(* CODESYS project OP60_PLC_program.project

Project tree, tasks and I/O mapping:
  Device : CODESYS Control Win V3 x64, 3S - Smart Software Solutions GmbH, version 3.5.16.40
    application Application
      libraries: VisuDialogs, * (System); MQTT Client SL, 1.0.2.0 (3S - Smart Software Solutions GmbH); SysTime, 3.5.9.0 (System); Util, * (System); StringUtils, 3.5.15.0 (System); Standard, * (System); SysFile, 3.5.15.0 (System)
      task MainTask (cyclic, interval t#20ms, priority 1) calls OP60_Main
      task AlarmManagerTask (cyclic, interval 50 ms, priority 1) calls AlarmManager.Alarm_Prg
      task VISU_TASK (cyclic, interval 100 ms, priority 1) calls VisuElems.Visu_Prg
      Symbols
      image pool ImagePool
      program SOP650 [LD]
      program OP60_Schedule [LD]
      FBs/
        function block FB_InputConveyor [LD]
        function block FB_SimpleConveyor [LD]
        function EraseSeconds [ST]
        program DateAndTime [ST]
        function TerminateString [ST]
        program CombineData [ST]
        function block FB_ModeControl [LD]
        function block FB_OutputConveyor [LD]
        function block FB_InspectionConveyor [LD]
        function Convert_RFID [ST]
      program SOP620 [LD]
      global variables GVL
      program OP60_Illumination [LD]
      program OP60_PublishMessages [LD]
      visualisation Production
      visualisation Overview
      program SOP690_GateEntry [LD]
      program OP60_Main [LD]
      program SOP600 [LD]
      program MQTTSub [ST]
      program SOP680 [LD]
      program SOP660 [LD]
      program Pruebas [LD]
      visualisation Manual_SOP640
      program SOP610 [LD]
      program SOP630 [LD]
      program OP60_Visu [LD]
      program MQTTPub [ST]
      visualisation Process
      visualisation Interfaces
      program SOP040_Safety [LD]
      global variables IOs
      Alarm Configuration
        alarm group SOP680_Alarms
            6814 [Fault]: Comparison Equal, ExpressionToCompare 14, Expression SOP680_FaultCode
            6805 [Fault]: Comparison Equal, ExpressionToCompare 5, Expression SOP680_FaultCode
            6811 [Fault]: Comparison Equal, ExpressionToCompare 11, Expression SOP680_FaultCode
            6802 [Fault]: Comparison Equal, ExpressionToCompare 2, Expression SOP680_FaultCode
            6812 [Fault]: Comparison Equal, ExpressionToCompare 12, Expression SOP680_FaultCode
            6810 [Fault]: Comparison Equal, ExpressionToCompare 10, Expression SOP680_FaultCode
            6801 [Fault]: Comparison Equal, ExpressionToCompare 1, Expression SOP680_FaultCode
            6813 [Fault]: Comparison Equal, ExpressionToCompare 13, Expression SOP680_FaultCode
        alarm class Fault (priority 10, acknowledge REP_ACK)
        alarm group SOP650_Alarms
            6512 [Fault]: Comparison Equal, ExpressionToCompare 12, Expression SOP650_FaultCode
            6514 [Fault]: Comparison Equal, ExpressionToCompare 14, Expression SOP650_FaultCode
            6501 [Fault]: Comparison Equal, ExpressionToCompare 1, Expression SOP650_FaultCode
            6511 [Fault]: Comparison Equal, ExpressionToCompare 11, Expression SOP650_FaultCode
            6510 [Fault]: Comparison Equal, ExpressionToCompare 10, Expression SOP650_FaultCode
            6505 [Fault]: Comparison Equal, ExpressionToCompare 5, Expression SOP650_FaultCode
            6513 [Fault]: Comparison Equal, ExpressionToCompare 13, Expression SOP650_FaultCode
            6502 [Fault]: Comparison Equal, ExpressionToCompare 2, Expression SOP650_FaultCode
        alarm group SOP660_Alarms
            6614 [Fault]: Comparison Equal, ExpressionToCompare 14, Expression SOP660_FaultCode
            6605 [Fault]: Comparison Equal, ExpressionToCompare 5, Expression SOP660_FaultCode
            6611 [Fault]: Comparison Equal, ExpressionToCompare 11, Expression SOP660_FaultCode
            6610 [Fault]: Comparison Equal, ExpressionToCompare 10, Expression SOP660_FaultCode
            6601 [Fault]: Comparison Equal, ExpressionToCompare 1, Expression SOP660_FaultCode
            6613 [Fault]: Comparison Equal, ExpressionToCompare 13, Expression SOP660_FaultCode
            6602 [Fault]: Comparison Equal, ExpressionToCompare 2, Expression SOP660_FaultCode
            6612 [Fault]: Comparison Equal, ExpressionToCompare 12, Expression SOP660_FaultCode
        alarm group SOP690_Alarms
            6901 [Fault]: Comparison Equal, ExpressionToCompare 0, Expression SOP690_NS1
            6902 [Fault]: Comparison Equal, ExpressionToCompare 0, Expression SOP690_B1
        alarm group SOP610_Alarms
            6110 [Fault]: Comparison Equal, ExpressionToCompare 10, Expression SOP610_FaultCode
            6101 [Fault]: Comparison Equal, ExpressionToCompare 1, Expression SOP610_FaultCode
            6111 [Fault]: Comparison Equal, ExpressionToCompare 11, Expression SOP610_FaultCode
            6114 [Fault]: Comparison Equal, ExpressionToCompare 14, Expression SOP610_FaultCode
            6105 [Fault]: Comparison Equal, ExpressionToCompare 5, Expression SOP610_FaultCode
            6113 [Fault]: Comparison Equal, ExpressionToCompare 13, Expression SOP610_FaultCode
            6102 [Fault]: Comparison Equal, ExpressionToCompare 2, Expression SOP610_FaultCode
            6112 [Fault]: Comparison Equal, ExpressionToCompare 12, Expression SOP610_FaultCode
        alarm group SOP670_Alarms
            6701 [Fault]: Comparison Equal, ExpressionToCompare 1, Expression SOP670_FaultCode
            6711 [Fault]: Comparison Equal, ExpressionToCompare 11, Expression SOP670_FaultCode
            6702 [Fault]: Comparison Equal, ExpressionToCompare 2, Expression SOP670_FaultCode
            6712 [Fault]: Comparison Equal, ExpressionToCompare 12, Expression SOP670_FaultCode
            6705 [Fault]: Comparison Equal, ExpressionToCompare 5, Expression SOP670_FaultCode
            6714 [Fault]: Comparison Equal, ExpressionToCompare 14, Expression SOP670_FaultCode
            6710 [Fault]: Comparison Equal, ExpressionToCompare 10, Expression SOP670_FaultCode
            6713 [Fault]: Comparison Equal, ExpressionToCompare 13, Expression SOP670_FaultCode
        alarm group SOP620_Alarms
            6205 [Fault]: Comparison Equal, ExpressionToCompare 5, Expression SOP620_FaultCode
            6202 [Fault]: Comparison Equal, ExpressionToCompare 2, Expression SOP620_FaultCode
            6212 [Fault]: Comparison Equal, ExpressionToCompare 12, Expression SOP620_FaultCode
            6201 [Fault]: Comparison Equal, ExpressionToCompare 1, Expression SOP620_FaultCode
            6211 [Fault]: Comparison Equal, ExpressionToCompare 11, Expression SOP620_FaultCode
            6213 [Fault]: Comparison Equal, ExpressionToCompare 13, Expression SOP620_FaultCode
            6210 [Fault]: Comparison Equal, ExpressionToCompare 10, Expression SOP620_FaultCode
            6214 [Fault]: Comparison Equal, ExpressionToCompare 14, Expression SOP620_FaultCode
        alarm group SOP600_Alarms
            6005 [Fault]: Comparison Equal, ExpressionToCompare 0, Expression SOP024_F12
            6003 [Fault]: Comparison Equal, ExpressionToCompare 0, Expression SOP024_F10
            6002 [Fault]: Comparison Equal, ExpressionToCompare 0, Expression SOP024_FQ1
            6008 [Fault]: Comparison Equal, ExpressionToCompare 0, Expression SOP040_B1
            6007 [Fault]: Comparison Equal, ExpressionToCompare 0, Expression SOP600_NS1
            6006 [Fault]: Comparison Equal, ExpressionToCompare 0, Expression SOP024_F13
            6004 [Fault]: Comparison Equal, ExpressionToCompare 0, Expression SOP024_F11
            6001 [Fault]: Comparison Equal, ExpressionToCompare 0, Expression SOP010_FQ1
        AlarmStorage
        alarm group SOP640_Alarms
            6402 [Fault]: Comparison Equal, ExpressionToCompare 2, Expression SOP640_FaultCode
            6412 [Fault]: Comparison Equal, ExpressionToCompare 12, Expression SOP640_FaultCode
            6422 [Fault]: Comparison Equal, ExpressionToCompare 22, Expression SOP640_FaultCode
            6410 [Fault]: Comparison Equal, ExpressionToCompare 10, Expression SOP640_FaultCode
            6414 [Fault]: Comparison Equal, ExpressionToCompare 14, Expression SOP640_FaultCode
            6413 [Fault]: Comparison Equal, ExpressionToCompare 13, Expression SOP640_FaultCode
            6420 [Fault]: Comparison Equal, ExpressionToCompare 20, Expression SOP640_FaultCode
            6430 [Fault]: Comparison Equal, ExpressionToCompare 0, Expression SOP640_LC1
            6405 [Fault]: Comparison Equal, ExpressionToCompare 5, Expression SOP640_FaultCode
            6401 [Fault]: Comparison Equal, ExpressionToCompare 1, Expression SOP640_FaultCode
            6411 [Fault]: Comparison Equal, ExpressionToCompare 11, Expression SOP640_FaultCode
            6421 [Fault]: Comparison Equal, ExpressionToCompare 21, Expression SOP640_FaultCode
            6423 [Fault]: Comparison Equal, ExpressionToCompare 23, Expression SOP640_FaultCode
        alarm class Warning (priority 30, acknowledge REP)
        text list TextList
        alarm group SOP630_Alarms
            6305 [Fault]: Comparison Equal, ExpressionToCompare 5, Expression SOP630_FaultCode
            6313 [Fault]: Comparison Equal, ExpressionToCompare 13, Expression SOP630_FaultCode
            6301 [Fault]: Comparison Equal, ExpressionToCompare 1, Expression SOP630_FaultCode
            6302 [Fault]: Comparison Equal, ExpressionToCompare 2, Expression SOP630_FaultCode
            6312 [Fault]: Comparison Equal, ExpressionToCompare 12, Expression SOP630_FaultCode
            6311 [Fault]: Comparison Equal, ExpressionToCompare 11, Expression SOP630_FaultCode
            6314 [Fault]: Comparison Equal, ExpressionToCompare 14, Expression SOP630_FaultCode
            6310 [Fault]: Comparison Equal, ExpressionToCompare 10, Expression SOP630_FaultCode
        alarm class Message (priority 100, acknowledge REP)
        alarm group OP60_Alarms
            0603 [Warning]: Comparison Equal, ExpressionToCompare 1, Expression OP60_ManDisInterlocks
            0601 [Message]: Comparison Equal, ExpressionToCompare 1, Expression OP60_WaitingToOP50
            0602 [Warning]: Comparison Equal, ExpressionToCompare 1, Expression OP60_EmptyMode
      program MQTT_Sensors_Actuators [LD]
      program SOP670 [LD]
      visualisation Diagnostics
      visualisation Manual_SOP610t630
      visualisation Manual_SOP650t680
      Cases/
        program Case1 [LD]
        program Case2 [LD]
        program Cases3_4_5 [LD]
      program SOP640 [LD]
  libraries: VisuSymbols, 3.5.10.0 (System)
  FuntionBlocks/
  5ce3da45-db07-42e7-a21c-a00fff4ed8f6|\\hsnas6\StaffHome\ayam\Documents\_MyStuff\13_Course AU334G\HMI\Motor Faulted.png
  visualisation Diagnostics
  5ce3da45-db07-42e7-a21c-a00fff4ed8f6|\\hsnas6\StaffHome\ayam\Documents\_MyStuff\13_Course AU334G\HMI\Door Open.png
  5ce3da45-db07-42e7-a21c-a00fff4ed8f6|\\hsnas6\StaffHome\ayam\Documents\_MyStuff\13_Course AU334G\HMI\Emergency Stop.png
  5ce3da45-db07-42e7-a21c-a00fff4ed8f6|\\hsnas6\StaffHome\ayam\Documents\_MyStuff\13_Course AU334G\HMI\Motor On.png
  5ce3da45-db07-42e7-a21c-a00fff4ed8f6|C:\Users\ayam\Dropbox\HiS\AUT02\Project\Layout.PNG
  5ce3da45-db07-42e7-a21c-a00fff4ed8f6|\\hsnas6\StaffHome\ayam\Documents\_MyStuff\13_Course AU334G\HMI\Motor Off.png
  text list GlobalTextList
  DataStructures/
    data type ProductionData
  text list System
  visualisation Production
  5ce3da45-db07-42e7-a21c-a00fff4ed8f6|\\hsnas6\StaffHome\ayam\Documents\_MyStuff\13_Course AU334G\HMI\Door Closed.png
*)

// DataStructures/ProductionData
TYPE ProductionData :
STRUCT
	ProductNr: UINT := 0; // Production Number
	IDNumber: UDINT := 0; // ID Number
	Status: WORD	:= 0; // Status Word
END_STRUCT
END_TYPE

// Device/Application/GVL
VAR_GLOBAL
	(* General *)
	Flash_1s: BOOL;		// Signal flashing (1Hz)
	Flash_2s: BOOL;		// Signal flashing (0.5Hz)
	Flash_2s_mem: BOOL;	// Flash_2s memory
	Client_Ready: BOOL;  // MQTT Ready
	ActualTime_hh_mm_ss: STRING; 		// Actual time HH:MM:SS format
	ActualTime_hh_mm: STRING;			// Actual time HH:MM:SS format
	Empty_PD : ProductionData;			// Empty Production Data
	
	Schedule_Start_msg: STRING(1024) := ''; 	// Received message from supervisor
	Schedule_End_msg: STRING(1024);		// Published message for supervisor
	Schedule_Start_msg_received: BOOL;		// Message is received again (this is made to avoid errors)
	Schedule_End_msg_received: BOOL; 			// Used to activate MQTT FB to publish message
	
	CycleData_Publish: BOOL; 				// Used to activate MQTT FB to publish message
	CycleData_pmsg: STRING(1024);			// Published message for further data analysis
	
	(* Light control should be in a sub-operation! *)
	Lights_msg: STRING(1024);			// Received message from supervisor/operator
	Lights_msg_received: BOOL;			// Message is received again (this is made to avoid errors)
	Switch_lights: BOOL;				// Used to activate turn on and off the lights
	Switch_msg: STRING(1024);			// Publish 'On' or 'Off' to turn on and off the lights
	Switch_publish: BOOL; 				// Order to publish
	Operator_pos_msg: STRING(1024);		// ????????????
	
	(* OP60 *)
	OP60_ModeControl: FB_ModeControl;
	OP60_Auto_On: BOOL; //OP60 in Auto-On
	OP60_Homing_On: BOOL; //OP60 in Homing-On
	OP60_Auto: BOOL; //OP60 in Auto Mode
	OP60_Manual: BOOL; // OP060 Manual Mode
	OP60_FaultAcc: BOOL; // OP60 Fault Accumulator
	OP60_WarningAcc: BOOL;	// OP60 Warning Accumulator
	OP60_SafetyCircuit_Ready: BOOL; // OP060 Safety Circuit Ready
	OP60_Stop_EOC_Req: BOOL; // OP060 Stop EOC Requested
	OP60_Stop_EOC_Ok: BOOL; // OP060 Stop EOC Ok
	OP60_HomePos_Ok: BOOL; // OP060 Home Position Ok
	OP60_ResetAlarms: BOOL; // OP60 Reset Alarms
	OP60_EOC AT %MW50: WORD; // OP060 EOC Word
	OP60_HomePos AT %MW51: WORD; // OP060 Home Pos Word
	OP60_ControlVoltage: BOOL; // Control Voltage Ready
	OP60_CtrlVoltageScheduleON: BOOL; // Control Voltage Schedule OFF
	OP60_CtrlVoltageScheduleOFF: BOOL; // Control Voltage Schedule ON
	OP60_WaitingToOP50: BOOL;	// OP60 Waiting to OP50
	OP60_WaitingToOP70: BOOL;	// OP60 Waiting to OP70
	OP60_ActualCycleTime: TIME; // Actual Cycle Time
	OP60_LastCycleTime: TIME; // Last Cycle Time
	OP60_TotalCycles: DWORD; // Total Cycles Counter
	OP60_EmptyMode: BOOL; // OP60 in Empty Mode
	OP60_ManDisInterlocks: BOOL; // OP060 Manual Mode
	OP60_ScheduleEnd: BOOL; // OP60 Schedule End
	OP60_ScheduleStart: BOOL; // OP60 Schedule Start
	HMI_DisableInterlocks: BOOL; // Disable Interlocks
	HMI_TotalCyclesReset: BOOL; //Total Cycles reset
	
	Operator_stop: BOOL;
	Operator_fault_msg: STRING(1024);
	Operator_fault_received: BOOL;
	
	SOP040_K1: BOOL;					// Safety Circuit OK
	SOP040_K1_msg: STRING(1024);		// OP60 Safety Circuit OK Message
	SOP040_K1_received: BOOL;			// Message is received again (this is made to avoid errors)
	SOP024_FQ1: BOOL;					// Power Suply Prim. Protection
	SOP024_FQ1_msg: STRING(1024);		// OP60 Power Suply Prim. Protection Message
	SOP024_FQ1_received: BOOL;			// Message is received again (this is made to avoid errors)
	SOP010_FQ1: BOOL;					// Supply Power Line Circuit Breaker
	SOP010_FQ1_msg: STRING(1024);		// OP60 Supply Power Line Circuit Breaker Message
	SOP010_FQ1_received: BOOL;			// Message is received again (this is made to avoid errors)
	SOP024_F10: BOOL;					// Power Suply Sec. Protection
	SOP024_F10_msg: STRING(1024);		// OP60 Power Suply Sec. Protection Message
	SOP024_F10_received: BOOL;			// Message is received again (this is made to avoid errors)
	SOP024_F11: BOOL;					// PLC Input Protection
	SOP024_F11_msg: STRING(1024);		// OP60 PLC Input Protection Message
	SOP024_F11_received: BOOL;			// Message is received again (this is made to avoid errors)
	SOP024_F12: BOOL;					// PLC Output Protection [HAY QUE QUITARLO]
	SOP024_F12_msg: STRING(1024);		// OP60 PLC Output Protection Message
	SOP024_F12_received: BOOL;			// Message is received again (this is made to avoid errors)
	SOP024_F13: BOOL;					// Safety Circuit Protection
	SOP024_F13_msg: STRING(1024);		// OP60 Safety Circuit Protection Message
	SOP024_F13_received: BOOL;			// Message is received again (this is made to avoid errors)
	SOP040_B1: BOOL;					// Pneumatic Pressure OK
	SOP040_B1_msg: STRING(1024);		// OP60 Pneumatic Pressure OK Message
	SOP040_B1_received: BOOL;			// Message is received again (this is made to avoid errors)
	
	(* OP50 Production Data *)
	OP50_PD : ProductionData;			// OP50 Last conveyor Production Data
	
	(* OP70 Production Data *)
	OP70_PD : ProductionData;			// OP70 First conveyor Production Data

	(* SOP600 *)
	SOP600_Faulted: BOOL;				// SOP600 Faulted
	
	SOP600_H1: BOOL;	// Control Voltage On Light
	SOP600_H2: BOOL; 	// Cycle Start Light
	SOP600_H3: BOOL;	// Cycle Stop Light
	SOP600_H4: BOOL; 	// Reset Alarm Light
	SOP600_H5: BOOL; 	// Reset Safety Light
	SOP600_H6: BOOL; 	// Blue Light
	SOP600_H7: BOOL; 	// Green Light
	SOP600_H8: BOOL; 	// Orange Light
	SOP600_H9: BOOL;	// Red Light
	SOP600_H10: BOOL;	// Home Position Light
	SOP600_H11: BOOL;	// Horn Sound
	
	SOP600_S1: BOOL;					// Control Voltage On
	SOP600_S1_msg: STRING(1024);		// SOP600_S1 Message
	SOP600_S1_received: BOOL;			// Message is received again (this is made to avoid errors)
	SOP600_S2: BOOL;					// Control Voltage Off
	SOP600_S2_msg: STRING(1024);		// SOP600_S2 Message
	SOP600_S2_received: BOOL;			// Message is received again (this is made to avoid errors)
	SOP600_S3: BOOL;					// Automatic Mode
	SOP600_S4: BOOL;					// Manual Mode
	SOP600_S3_4: BOOL;					// Automatic and Manual Mode
	SOP600_S3_4_msg: STRING(1024);		// SOP600_S4 Message
	SOP600_S3_4_received: BOOL;			// Message is received again (this is made to avoid errors)
	SOP600_S5: BOOL;					// Cycle Start
	SOP600_S5_msg: STRING(1024);		// SOP600_S5 Message
	SOP600_S5_received: BOOL;			// Message is received again (this is made to avoid errors)
	SOP600_S6: BOOL;					// Cycle Stop
	SOP600_S6_msg: STRING(1024);		// SOP600_S6 Message
	SOP600_S6_received: BOOL;			// Message is received again (this is made to avoid errors)
	SOP600_S7: BOOL;					// Halt
	SOP600_S7_msg: STRING(1024);		// SOP600_S7 Message
	SOP600_S7_received: BOOL;			// Message is received again (this is made to avoid errors)
	SOP600_S8: BOOL;					// Reset Alarm
	SOP600_S8_msg: STRING(1024);		// SOP600_S8 Message
	SOP600_S8_received: BOOL;			// Message is received again (this is made to avoid errors)
	SOP600_S9: BOOL;					// Reset Safety
	SOP600_S9_msg: STRING(1024);		// SOP600_S9 Message
	SOP600_S9_received: BOOL;			// Message is received again (this is made to avoid errors)
	SOP600_S10: BOOL;					// Home Position
	SOP600_S10_msg: STRING(1024);		// SOP600_S10 Message
	SOP600_S10_received: BOOL;			// Message is received again (this is made to avoid errors)
	SOP600_S11: BOOL;					// Emergency Stop
	SOP600_S11_msg: STRING(1024);		// SOP600_S11 Message
	SOP600_S11_received: BOOL;			// Message is received again (this is made to avoid errors)
	
	SOP040_K3: BOOL;					// Reset Safety circuit
	SOP040_K3_pmsg: STRING(1024);			// Published message for the logics
	SOP040_K3_publish: BOOL;				// Used to activate MQTT FB to publish message
	SOP600_H6_pmsg: STRING(1024);			// Published message for the logics
	SOP600_H6_publish: BOOL;				// Used to activate MQTT FB to publish message
	SOP600_H7_pmsg: STRING(1024);			// Published message for the logics
	SOP600_H7_publish: BOOL;				// Used to activate MQTT FB to publish message
	SOP600_H8_pmsg: STRING(1024);			// Published message for the logics
	SOP600_H8_publish: BOOL;				// Used to activate MQTT FB to publish message
	SOP600_H9_pmsg: STRING(1024);			// Published message for the logics
	SOP600_H9_publish: BOOL;				// Used to activate MQTT FB to publish message
	SOP600_S1_pmsg: STRING(1024);			// Published message for the logics
	SOP600_S1_publish: BOOL;				// Used to activate MQTT FB to publish message
	SOP600_S5_pmsg: STRING(1024);			// Published message for the logics
	SOP600_S5_publish: BOOL;				// Used to activate MQTT FB to publish message
	SOP600_S6_pmsg: STRING(1024);			// Published message for the logics
	SOP600_S6_publish: BOOL;				// Used to activate MQTT FB to publish message
	SOP600_S8_pmsg: STRING(1024);			// Published message for the logics
	SOP600_S8_publish: BOOL;				// Used to activate MQTT FB to publish message
	SOP600_S9_pmsg: STRING(1024);			// Published message for the logics
	SOP600_S9_publish: BOOL;				// Used to activate MQTT FB to publish message
	SOP600_S10_pmsg: STRING(1024);			// Published message for the logics
	SOP600_S10_publish: BOOL;				// Used to activate MQTT FB to publish message
	SOP600_S11_pmsg: STRING(1024);			// Published message for the logics
	SOP600_S11_publish: BOOL;				// Used to activate MQTT FB to publish message
	
	(* SOP610 *)
	SOP610_Conveyor: FB_InputConveyor; // SOP610_Conveyor
	SOP610_PD: ProductionData; 			// SOP610 Production Data
	SOP610_Faulted: BOOL;				// SOP610 Faulted
	SOP610_FaultCode: INT;				// SOP610 Fault Code
	SOP610_EOC AT %MX100.0: BOOL;		// SOP610 At EOC
	SOP610_HomePos AT %MX102.0: BOOL;	// SOP610 At Home Position
	
	SOP610_ReadyToTransfer: BOOL; 		// SOP610 Conveyor ready to transfer
	SOP610_Transfering: BOOL; 			// SOP610 Conveyor transfering
	SOP610_MovePD: BOOL;				// SOP610 Move Production Data
	
	HMI_SOP610_ManMoveFwd: BOOL; 		// SOP610 Manual Move Conveyor Fwd 
	HMI_SOP610_ManMoveRev: BOOL; 		// SOP610 Manual Move Conveyor Rev 
	HMI_SOP610_ManPDFwd: BOOL; 			// SOP610 Manual Move Production Data Fwd 
	HMI_SOP610_ManPDRev: BOOL; 			// SOP610 Manual Move Production Data Rev 
	
	SOP610_B1: BOOL;					// Conveyor Sensor
	SOP610_B1_msg: STRING(1024);		// SOP610 Photoelectric Sensor Message
	SOP610_B1_received: BOOL;			// Message is received again (this is made to avoid errors)
	SOP610_FQ1: BOOL;					// Motor Protection Tripped
	SOP610_FQ1_msg: STRING(1024);		// SOP610 Motor Protection Tripped Message
	SOP610_FQ1_received: BOOL;			// Message is received again (this is made to avoid errors)
	SOP610_RFID_Read: INT;							// RFID Read 
	SOP610_RFID_Read_msg: STRING(1024);				// SOP610 RFID Read Message
	SOP610_RFID_Read_received: BOOL;				// Message is received again (this is made to avoid errors)
	SOP610_RFID_Status: INT;						// RFID Status
	SOP610_RFID_Status_msg: STRING(1024);			// SOP610 RFID Status Message
	SOP610_RFID_Status_received: BOOL;				// Message is received again (this is made to avoid errors)
	
	// SOP610_RFID_Control: INT;				// RFID Contol
	SOP610_RFID_Control_pmsg: STRING(1024);	// Published message for the logics
	SOP610_RFID_Control_publish: BOOL;		// FB is publishing message
	// SOP610_RFID_Write: STRING;				// RFID Write
	SOP610_RFID_Write_pmsg: STRING(1024);	// Published message for the logics
	SOP610_RFID_Write_publish: BOOL;		// FB is publishing message
	SOP610_KM1: BOOL;						// Conveyor Forward
	SOP610_KM2: BOOL;						// Conveyor Reverse
	SOP610_KM1_2_pmsg: STRING(1024);		// Published message for the logics
	SOP610_KM1_2_pbusy: BOOL;				// FB is publishing message
	SOP610_KM1_2_publish: BOOL;				// Used to activate MQTT FB to publish message

	(* SOP620 *)
	SOP620_Conveyor: FB_SimpleConveyor; // SOP620_Conveyor
	SOP620_PD: ProductionData; 			// SOP620 Production Data
	SOP620_Faulted: BOOL;				// SOP620 Faulted
	SOP620_FaultCode: INT;				// SOP620 Fault Code
	SOP620_EOC AT %MX100.1: BOOL;		// SOP620 At EOC
	SOP620_HomePos AT %MX102.1: BOOL;	// SOP620 At Home Position
	
	SOP620_ReadyToTransfer: BOOL; 		// SOP620 Conveyor ready to transfer
	SOP620_Transfering: BOOL; 			// SOP620 Conveyor transfering
	SOP620_TransferOK: BOOL; 			// SOP620 Conveyor ready to load
	SOP620_TransferDone: BOOL; 			// SOP620 Conveyor load completed
	SOP620_MovePD: BOOL;				// SOP620 Move Production Data
	
	HMI_SOP620_ManMoveFwd: BOOL; 		// SOP620 Manual Move Conveyor Fwd 
	HMI_SOP620_ManMoveRev: BOOL; 		// SOP620 Manual Move Conveyor Rev 
	HMI_SOP620_ManPDFwd: BOOL; 			// SOP620 Manual Move Production Data Fwd 
	HMI_SOP620_ManPDRev: BOOL; 			// SOP620 Manual Move Production Data Rev 
	
	SOP620_B1: BOOL;					// Conveyor Sensor
	SOP620_B1_msg: STRING(1024);				// SOP620 Photoelectric Sensor Message
	SOP620_B1_received: BOOL;			// Message is received again (this is made to avoid errors)
	SOP620_FQ1: BOOL;					// Motor Protection Tripped
	SOP620_FQ1_msg: STRING(1024);		// SOP620 Motor Protection Tripped Message
	SOP620_FQ1_received: BOOL;			// Message is received again (this is made to avoid errors)
	
	SOP620_KM1: BOOL;						// Conveyor Forward
	SOP620_KM2: BOOL;						// Conveyor Reverse
	SOP620_KM1_2_pmsg: STRING(1024);		// Published message for the logics
	SOP620_KM1_2_pbusy: BOOL;				// FB is publishing message
	SOP620_KM1_2_publish: BOOL;				// Used to activate MQTT FB to publish message
	
	(* SOP630 *)
	SOP630_Conveyor: FB_SimpleConveyor; // SOP630_Conveyor
	SOP630_PD: ProductionData; 			// SOP630 Production Data
	SOP630_Faulted: BOOL;				// SOP630 Faulted
	SOP630_FaultCode: INT;				// SOP630 Fault Code
	SOP630_EOC AT %MX100.2: BOOL;		// SOP630 At EOC
	SOP630_HomePos AT %MX102.2: BOOL;	// SOP630 At Home Position
	
	SOP630_ReadyToTransfer: BOOL; 		// SOP630 Conveyor ready to transfer
	SOP630_Transfering: BOOL; 			// SOP630 Conveyor transfering
	SOP630_TransferOK: BOOL; 			// SOP630 Conveyor ready to load
	SOP630_TransferDone: BOOL; 			// SOP630 Conveyor load completed
	SOP630_MovePD: BOOL;				// SOP630 Move Production Data
	
	HMI_SOP630_ManMoveFwd: BOOL; 		// SOP630 Manual Move Conveyor Fwd 
	HMI_SOP630_ManMoveRev: BOOL; 		// SOP630 Manual Move Conveyor Rev 
	HMI_SOP630_ManPDFwd: BOOL; 			// SOP630 Manual Move Production Data Fwd 
	HMI_SOP630_ManPDRev: BOOL; 			// SOP630 Manual Move Production Data Rev 
	
	SOP630_B1: BOOL;					// Conveyor Sensor
	SOP630_B1_msg: STRING(1024);		// SOP630 Photoelectric Sensor Message
	SOP630_B1_received: BOOL;			// Message is received again (this is made to avoid errors)
	SOP630_FQ1: BOOL;					// Motor Protection Tripped
	SOP630_FQ1_msg: STRING(1024);		// SOP630 Motor Protection Tripped Message
	SOP630_FQ1_received: BOOL;			// Message is received again (this is made to avoid errors)
	
	SOP630_KM1: BOOL;						// Conveyor Forward
	SOP630_KM2: BOOL;						// Conveyor Reverse
	SOP630_KM1_2_pmsg: STRING(1024);		// Published message for the logics
	SOP630_KM1_2_pbusy: BOOL;				// FB is publishing message
	SOP630_KM1_2_publish: BOOL;				// Used to activate MQTT FB to publish message

	(* SOP640 *)
	SOP640_Conveyor: FB_InspectionConveyor; // SOP640_Conveyor
	SOP640_PD: ProductionData; 			// SOP640 Production Data
	SOP640_Faulted: BOOL;				// SOP640 Faulted
	SOP640_FaultCode: INT;				// SOP640 Fault Code
	SOP640_EOC AT %MX100.3: BOOL;		// SOP640 At EOC
	SOP640_HomePos AT %MX102.3: BOOL;	// SOP640 At Home Position
	
	SOP640_ReadyToTransfer: BOOL; 		// SOP640 Conveyor ready to transfer
	SOP640_Transfering: BOOL; 			// SOP640 Conveyor transfering
	SOP640_TransferOK: BOOL; 			// SOP640 Conveyor ready to load
	SOP640_TransferDone: BOOL; 			// SOP640 Conveyor load completed
	SOP640_MovePD: BOOL;				// SOP640 Move Production Data
	
	HMI_SOP640_ManMoveFwd: BOOL; 		// SOP640 Manual Move Conveyor Fwd 
	HMI_SOP640_ManMoveRev: BOOL; 		// SOP640 Manual Move Conveyor Rev 
	HMI_SOP640_ManFrontUp: BOOL;		// SOP640 Manual Move Front Clamp Up 
	HMI_SOP640_ManFrontDown: BOOL;		// SOP640 Manual Move Front Clamp Down
	HMI_SOP640_ManRearUp: BOOL;			// SOP640 Manual Move Rear Clamp Up
	HMI_SOP640_ManRearDown: BOOL;		// SOP640 Manual Move Rear Clamp Down
	HMI_SOP640_ManPDFwd: BOOL; 			// SOP640 Manual Move Production Data Fwd 
	HMI_SOP640_ManPDRev: BOOL; 			// SOP640 Manual Move Production Data Rev 
	HMI_SOP640_Accept: BOOL;			// SOP640 Accept Inspection
	HMI_SOP640_Discard: BOOL;			// SOP640 Discard Inspection
	HMI_SOP640_Inspecting: BOOL;		// SOP640 Discard Inspection
	
	SOP640_RS: BOOL;
	
	SOP640_Publish: BOOL; 				// Used to activate MQTT FB to publish message
	SOP640_pmsg: STRING(4096);			// Published message for operator
	SOP640_A1: BOOL;					// Conveyor Sensor
	SOP640_A1_msg: STRING(1024);		// SOP650 Photoelectric Sensor Message
	SOP640_A1_received: BOOL;			// Message is received again (this is made to avoid errors)
	SOP640_B1: BOOL;					// Conveyor Sensor
	SOP640_B1_msg: STRING(1024);				// SOP640 Photoelectric Sensor Message
	SOP640_B1_received: BOOL;			// Message is received again (this is made to avoid errors)
	SOP640_B2: BOOL(1024);					// Cylinder Sensor
	SOP640_B2_msg: STRING(1024);				// SOP640 Photoelectric Sensor Message
	SOP640_B2_received: BOOL;			// Message is received again (this is made to avoid errors)
	SOP640_B3: BOOL;					// Cylinder Sensor
	SOP640_B3_msg: STRING(1024);				// SOP640 Photoelectric Sensor Message
	SOP640_B3_received: BOOL;			// Message is received again (this is made to avoid errors)
	SOP640_B4: BOOL;					// Cylinder Sensor
	SOP640_B4_msg: STRING(1024);				// SOP640 Photoelectric Sensor Message
	SOP640_B4_received: BOOL;			// Message is received again (this is made to avoid errors)
	SOP640_B5: BOOL;					// Cylinder Sensor
	SOP640_B5_msg: STRING(1024);				// SOP640 Photoelectric Sensor Message
	SOP640_B5_received: BOOL;			// Message is received again (this is made to avoid errors)
	SOP640_B6: BOOL;					// Proximity Sensor
	SOP640_B6_msg: STRING(1024);				// SOP640 Photoelectric Sensor Message
	SOP640_B6_received: BOOL;			// Message is received again (this is made to avoid errors)
	SOP640_FQ1: BOOL;					// Motor Protection Tripped
	SOP640_FQ1_msg: STRING(1024);		// SOP640 Motor Protection Tripped Message
	SOP640_FQ1_received: BOOL;			// Message is received again (this is made to avoid errors)
	
	SOP640_KM1: BOOL;						// Conveyor Forward
	SOP640_KM2: BOOL;						// Conveyor Reverse
	SOP640_KM1_2_pmsg: STRING(1024);		// Published message for the logics
	SOP640_KM1_2_pbusy: BOOL;				// FB is publishing message
	SOP640_KM1_2_publish: BOOL;				// Used to activate MQTT FB to publish message
	SOP640_K2: BOOL;						// Stopper Up
	SOP640_K2_pmsg: STRING(1024);			// Published message for the logics
	SOP640_K2_publish: BOOL;				// Used to activate MQTT FB to publish message
	SOP640_Y1: BOOL;						// Stopper Up
	SOP640_Y1_pmsg: STRING(1024);			// Published message for the logics
	SOP640_Y1_publish: BOOL;				// Used to activate MQTT FB to publish message
	SOP640_Y2: BOOL;						// Stopper Down
	SOP640_Y2_pmsg: STRING(1024);			// Published message for the logics
	SOP640_Y2_publish: BOOL;				// Used to activate MQTT FB to publish message
	SOP640_Y3: BOOL;						// Stopper Up
	SOP640_Y3_pmsg: STRING(1024);			// Published message for the logics
	SOP640_Y3_publish: BOOL;				// Used to activate MQTT FB to publish message
	SOP640_Y4: BOOL;						// Stopper Down
	SOP640_Y4_pmsg: STRING(1024);			// Published message for the logics
	SOP640_Y4_publish: BOOL;				// Used to activate MQTT FB to publish message
	Products_publish: BOOL;					// Products data
	Products_pmsg: STRING(1024);			// Publish message for the logics
	
	// SOP640_RFID_Control: INT;				// RFID Contol
	SOP640_RFID_Control_pmsg: STRING(1024);	// Published message for the logics
	SOP640_RFID_Control_publish: BOOL;		// FB is publishing message
	// SOP640_RFID_Write: STRING;				// RFID Write
	SOP640_RFID_Write_pmsg: STRING(1024);	// Published message for the logics
	SOP640_RFID_Write_publish: BOOL;		// FB is publishing message
	
	Inspection_msg: STRING(1024) := ''; // Received message from SOP640 operator
	Inspection_msg_received: BOOL;		// Message is received again (this is made to avoid previous product status)

	(* SOP650 *)
	SOP650_Conveyor: FB_SimpleConveyor; // SOP650_Conveyor
	SOP650_PD: ProductionData; 			// SOP650 Production Data
	SOP650_Faulted: BOOL;				// SOP650 Faulted
	SOP650_FaultCode: INT;				// SOP650 Fault Code
	SOP650_EOC AT %MX100.4: BOOL;		// SOP650 At EOC
	SOP650_HomePos AT %MX102.4: BOOL;	// SOP650 At Home Position
	
	SOP650_ReadyToTransfer: BOOL; 		// SOP650 Conveyor ready to transfer
	SOP650_Transfering: BOOL; 			// SOP650 Conveyor transfering
	SOP650_TransferOK: BOOL; 			// SOP650 Conveyor ready to load
	SOP650_TransferDone: BOOL; 			// SOP650 Conveyor load completed
	SOP650_MovePD: BOOL;				// SOP650 Move Production Data
	
	HMI_SOP650_ManMoveFwd: BOOL; 		// SOP650 Manual Move Conveyor Fwd 
	HMI_SOP650_ManMoveRev: BOOL; 		// SOP650 Manual Move Conveyor Rev 
	HMI_SOP650_ManPDFwd: BOOL; 			// SOP650 Manual Move Production Data Fwd 
	HMI_SOP650_ManPDRev: BOOL; 			// SOP650 Manual Move Production Data Rev 
	
	
	SOP650_B1: BOOL;					// Conveyor Sensor
	SOP650_B1_msg: STRING(1024);		// SOP650 Photoelectric Sensor Message
	SOP650_B1_received: BOOL;			// Message is received again (this is made to avoid errors)
	SOP650_FQ1: BOOL;					// Motor Protection Tripped
	SOP650_FQ1_msg: STRING(1024);		// SOP610 Motor Protection Tripped Message
	SOP650_FQ1_received: BOOL;			// Message is received again (this is made to avoid errors)
	
	SOP650_KM1: BOOL;						// Conveyor Forward
	SOP650_KM2: BOOL;						// Conveyor Reverse
	SOP650_KM1_2_pbusy: BOOL;				// FB is publishing message
	SOP650_KM1_2_pmsg: STRING(1024);		// Published message for the logics
	SOP650_KM1_2_publish: BOOL;				// Used to activate MQTT FB to publish message

	(* SOP660 *)
	SOP660_Conveyor: FB_SimpleConveyor; // SOP660_Conveyor
	SOP660_PD: ProductionData; 			// SOP660 Production Data
	SOP660_Faulted: BOOL;				// SOP660 Faulted
	SOP660_FaultCode: INT;				// SOP660 Fault Code
	SOP660_EOC AT %MX100.5: BOOL;		// SOP660 At EOC
	SOP660_HomePos AT %MX102.5: BOOL;	// SOP660 At Home Position
	
	SOP660_ReadyToTransfer: BOOL; 		// SOP660 Conveyor ready to transfer
	SOP660_Transfering: BOOL; 			// SOP660 Conveyor transfering
	SOP660_TransferOK: BOOL; 			// SOP660 Conveyor ready to load
	SOP660_TransferDone: BOOL; 			// SOP660 Conveyor load completed
	SOP660_MovePD: BOOL;				// SOP660 Move Production Data
	
	HMI_SOP660_ManMoveFwd: BOOL; 		// SOP660 Manual Move Conveyor Fwd 
	HMI_SOP660_ManMoveRev: BOOL; 		// SOP660 Manual Move Conveyor Rev 
	HMI_SOP660_ManPDFwd: BOOL; 			// SOP660 Manual Move Production Data Fwd 
	HMI_SOP660_ManPDRev: BOOL; 			// SOP660 Manual Move Production Data Rev 
	
	SOP660_B1: BOOL;					// Conveyor Sensor
	SOP660_B1_msg: STRING(1024);		// SOP660 Photoelectric Sensor Message
	SOP660_B1_received: BOOL;			// Message is received again (this is made to avoid errors)
	SOP660_FQ1: BOOL;					// Motor Protection Tripped
	SOP660_FQ1_msg: STRING(1024);		// SOP660 Motor Protection Tripped Message
	SOP660_FQ1_received: BOOL;			// Message is received again (this is made to avoid errors)
	
	SOP660_KM1: BOOL;						// Conveyor Forward
	SOP660_KM2: BOOL;						// Conveyor Reverse
	SOP660_KM1_2_pbusy: BOOL;				// FB is publishing message
	SOP660_KM1_2_pmsg: STRING(1024);		// Published message for the logics
	SOP660_KM1_2_publish: BOOL;				// Used to activate MQTT FB to publish message

	(* SOP670 *)
	SOP670_Conveyor: FB_SimpleConveyor; // SOP670_Conveyor
	SOP670_PD: ProductionData; 			// SOP670 Production Data
	SOP670_Faulted: BOOL;				// SOP670 Faulted
	SOP670_FaultCode: INT;				// SOP670 Fault Code
	SOP670_EOC AT %MX100.6: BOOL;		// SOP670 At EOC
	SOP670_HomePos AT %MX102.6: BOOL;	// SOP670 At Home Position
	
	SOP670_ReadyToTransfer: BOOL; 		// SOP670 Conveyor ready to transfer
	SOP670_Transfering: BOOL; 			// SOP670 Conveyor transfering
	SOP670_TransferOK: BOOL; 			// SOP670 Conveyor ready to load
	SOP670_TransferDone: BOOL; 			// SOP670 Conveyor load completed
	SOP670_MovePD: BOOL;				// SOP670 Move Production Data
	
	HMI_SOP670_ManMoveFwd: BOOL; 		// SOP670 Manual Move Conveyor Fwd 
	HMI_SOP670_ManMoveRev: BOOL; 		// SOP670 Manual Move Conveyor Rev 
	HMI_SOP670_ManPDFwd: BOOL; 			// SOP670 Manual Move Production Data Fwd 
	HMI_SOP670_ManPDRev: BOOL; 			// SOP670 Manual Move Production Data Rev 
	
	SOP670_KM1: BOOL;						// Conveyor Forward
	SOP670_KM2: BOOL;						// Conveyor Reverse
	SOP670_KM1_2_pbusy: BOOL;				// FB is publishing message
	SOP670_B1: BOOL;					// Conveyor Sensor
	SOP670_B1_msg: STRING(1024);		// SOP670 Photoelectric Sensor Message
	SOP670_B1_received: BOOL;			// Message is received again (this is made to avoid errors)
	SOP670_FQ1: BOOL;					// Motor Protection Tripped
	SOP670_FQ1_msg: STRING(1024);		// SOP670 Motor Protection Tripped Message
	SOP670_FQ1_received: BOOL;			// Message is received again (this is made to avoid errors)
	
	SOP670_KM1_2_pmsg: STRING(1024);		// Published message for the logics
	SOP670_KM1_2_publish: BOOL;				// Used to activate MQTT FB to publish message

	(* SOP680 *)
	SOP680_Conveyor: FB_OutputConveyor; // SOP680_Conveyor
	SOP680_PD: ProductionData; 			// SOP680 Production Data
	SOP680_Faulted: BOOL;				// SOP680 Faulted
	SOP680_FaultCode: INT;				// SOP680 Fault Code
	SOP680_EOC AT %MX100.7: BOOL;		// SOP680 At EOC
	SOP680_HomePos AT %MX102.7: BOOL;	// SOP680 At Home Position
	
	SOP680_TransferOK: BOOL; 			// SOP680 Conveyor ready to load
	SOP680_TransferDone: BOOL; 			// SOP680 Conveyor load completed
	SOP680_MovePD: BOOL;				// SOP680 Move Production Data
	
	HMI_SOP680_ManMoveFwd: BOOL; 		// SOP680 Manual Move Conveyor Fwd 
	HMI_SOP680_ManMoveRev: BOOL; 		// SOP680 Manual Move Conveyor Rev 
	HMI_SOP680_ManPDFwd: BOOL; 			// SOP680 Manual Move Production Data Fwd 
	HMI_SOP680_ManPDRev: BOOL; 			// SOP680 Manual Move Production Data Rev 
	
	SOP680_B1: BOOL;					// Conveyor Sensor
	SOP680_B1_msg: STRING(1024);		// SOP680 Photoelectric Sensor Message
	SOP680_B1_received: BOOL;			// Message is received again (this is made to avoid errors)
	SOP680_FQ1: BOOL;					// Motor Protection Tripped
	SOP680_FQ1_msg: STRING(1024);		// SOP680 Motor Protection Tripped Message
	SOP680_FQ1_received: BOOL;			// Message is received again (this is made to avoid errors)
	
	SOP680_KM1: BOOL;						// Conveyor Forward
	SOP680_KM2: BOOL;						// Conveyor Reverse
	SOP680_KM1_2_pbusy: BOOL;				// FB is publishing message
	SOP680_KM1_2_pmsg: STRING(1024);		// Published message for the logics
	SOP680_KM1_2_publish: BOOL;				// Used to activate MQTT FB to publish message

	(* SOP690 *)
	SOP690_EntryRequest: BOOL;			// SOP690 Entry Request
	SOP690_Faulted: BOOL;				// SOP690 Faulted
	
	SOP690_K1: BOOL; 					// Gate Unlocked Confirmation
	SOP690_S1: BOOL;					// Cycle Start
	SOP690_S1_msg: STRING(1024);		// SOP690_S1 Message
	SOP690_S1_received: BOOL;			// Message is received again (this is made to avoid errors)
	SOP690_S2: BOOL;					// Entry Request
	SOP690_S2_msg: STRING(1024);		// SOP690_S2 Message
	SOP690_S2_received: BOOL;			// Message is received again (this is made to avoid errors)
	SOP690_S3: BOOL;					// Emergency Stop
	SOP690_S3_msg: STRING(1024);		// SOP690_S3 Message
	SOP690_S3_received: BOOL;			// Message is received again (this is made to avoid errors)
	SOP690_B1: BOOL;					// Gate Closed
	SOP690_S4: BOOL;					// Unlock Gate
	SOP690_S4_msg: STRING(1024);		// SOP690_S4 Message
	SOP690_S4_received: BOOL;			// Message is received again (this is made to avoid errors)

	SOP690_H1: BOOL;					// Cycle Start Light
	SOP690_H2: BOOL;					// Entry Request Light
	SOP690_H3: BOOL;					// Reset Safety Light
	
	SOP690_S1_pmsg: STRING(1024);			// Published message for the logics
	SOP690_S1_publish: BOOL;				// Used to activate MQTT FB to publish message
	SOP690_S2_pmsg: STRING(1024);			// Published message for the logics
	SOP690_S2_publish: BOOL;				// Used to activate MQTT FB to publish message
	SOP690_S3_pmsg: STRING(1024);			// Published message for the logics
	SOP690_S3_publish: BOOL;				// Used to activate MQTT FB to publish message
	SOP690_S4_pmsg: STRING(1024);			// Published message for the logics
	SOP690_S4_publish: BOOL;				// Used to activate MQTT FB to publish message
	
	SOP690_RFID_Read: INT;							// RFID Read 
	SOP690_RFID_Read_msg: STRING(1024);				// SOP690 RFID Read Message
	SOP690_RFID_Read_received: BOOL;				// Message is received again (this is made to avoid errors)
	SOP690_RFID_Status: INT;						// RFID Status
	SOP690_RFID_Status_msg: STRING(1024);			// SOP690 RFID Status Message
	SOP690_RFID_Status_received: BOOL;				// Message is received again (this is made to avoid errors)
	// SOP690_RFID_Control: INT;					// RFID Contol
	SOP690_RFID_Control_pmsg: STRING(1024);			// Published message for the logics
	SOP690_RFID_Control_publish: BOOL;				// FB is publishing message
END_VAR

// Device/Application/IOs
VAR_GLOBAL
	(* INPUTS*) 
	//Name	Address	Type	Comment
	SOP004_A1_4	AT %MW0	: WORD;	// 16 DI Card, Input 0-7 
	//1 SOP010_FQ1	AT %MX0.0	: BOOL;	// Supply Power Line Circuit Breaker
	//2 SOP040_K1	AT %MX0.1	: BOOL;	// Safety Circuit OK
	//3 SOP024_FQ1	AT %MX0.2	: BOOL;	// Power Suply Prim. Protection
	//4 SOP024_F10	AT %MX0.3	: BOOL;	// Power Suply Sec. Protection
	//5 SOP024_F11	AT %MX0.4	: BOOL;	// PLC Input Protection
	//6 SOP024_F12	AT %MX0.5	: BOOL;	// PLC Output Protection
	//7 SOP024_F13	AT %MX0.6	: BOOL;	// Safety Circuit Protection
	//8 SOP040_B1	AT %MX0.7	: BOOL;	// Pneumatic Pressure OK
	//SOP004_A1_4_2	AT %MB1	: BYTE;	// 16 DI Card, Input 8-15 
	M16_Entry	AT %MX1.0	: BOOL;	// 
	M16T_Entry	AT %MX1.1	: BOOL;	// 
	M20_Entry	AT %MX1.2	: BOOL;	// 
	M24_Entry	AT %MX1.3	: BOOL;	// 
	//Reserved	AT %MX1.4	: BOOL;	// 
	//Reserved	AT %MX1.5	: BOOL;	// 
	//Reserved	AT %MX1.6	: BOOL;	// 
	//Reserved	AT %MX1.7	: BOOL;	// 
	SOP004_A1_5	AT %MW1	: WORD;	// 16 DI Card, Input 0-7 
	//9 SOP600_S1	AT %MX2.0	: BOOL;	// Control Voltage On
	//10 SOP600_S2	AT %MX2.1	: BOOL;	// Control Voltage Off
	//11 SOP600_S3	AT %MX2.2	: BOOL;	// Manual Mode
	//12 SOP600_S4	AT %MX2.3	: BOOL;	// Automatic Mode
	//13 SOP600_S5	AT %MX2.4	: BOOL;	// Cycle Start
	//14 SOP600_S6	AT %MX2.5	: BOOL;	// Cycle Stop
	//15 SOP600_S7	AT %MX2.6	: BOOL;	// Halt
	//16 SOP600_S8	AT %MX2.7	: BOOL;	// Reset Alarm
	//SOP004_A1_5_2	AT %MB3	: BYTE;	// 16 DI Card, Input 8-15 
	//17 SOP600_S9	AT %MX3.0	: BOOL;	// Reset Safety
	//18 SOP600_S10	AT %MX3.1	: BOOL;	// Home Position     (* SOP600_S11 NOT DEFINED? *)
	SOP600_NS1	AT %MX3.2	: BOOL;	// Emergency Stop
	//Reserved	AT %MX3.3	: ;	// 
	//Reserved	AT %MX3.4	: ;	// 
	//Reserved	AT %MX3.5	: ;	// 
	//Reserved	AT %MX3.6	: ;	// 
	//Reserved	AT %MX3.7	: ;	// 
	SOP004_A1_6	AT %MW2	: WORD;	// 16 DI Card, Input 0-7 
	//19 SOP610_FQ1	AT %MX4.0	: BOOL;	// Motor Protection Tripped
	//20 SOP610_B1	AT %MX4.1	: BOOL;	// Conveyor Sensor
	//21 SOP620_FQ1	AT %MX4.2	: BOOL;	// Motor Protection Tripped
	//22 SOP620_B1	AT %MX4.3	: BOOL;	// Conveyor Sensor
	//23 SOP630_FQ1	AT %MX4.4	: BOOL;	// Motor Protection Tripped
	//24 SOP630_B1	AT %MX4.5	: BOOL;	// Conveyor Sensor
	//Reserved	AT %MX4.6	: ;	// 
	//Reserved	AT %MX4.7	: ;	// 
	//SOP004_A1_6_2	AT %MB5	: BYTE;	// 16 DI Card, Input 8-15 
	//25 SOP640_FQ1	AT %MX5.0	: BOOL;	// Motor Protection Tripped
	//26 SOP640_B1	AT %MX5.1	: BOOL;	// Conveyor Sensor
	//27 SOP640_B2	AT %MX5.2	: BOOL;	// Front Clamp Down
	//28 SOP640_B3	AT %MX5.3	: BOOL;	// Front Clamp Up
	//29 SOP640_B4	AT %MX5.4	: BOOL;	// Rear Clamp Down
	//30 SOP640_B5	AT %MX5.5	: BOOL;	// Rear Clamp Up
	//31 SOP640_B6	AT %MX5.6	: BOOL;	// Operator Proximity Sensor 
	SOP640_LC1	AT %MX5.7	: BOOL;	// Light Curtain OK
	SOP004_A1_7	AT %MW3	: WORD;	// 16 DI Card, Input 0-7 
	//33 SOP650_FQ1	AT %MX6.0	: BOOL;	// Motor Protection Tripped
	//34 SOP650_B1	AT %MX6.1	: BOOL;	// Conveyor Sensor
	//35 SOP660_FQ1	AT %MX6.2	: BOOL;	// Motor Protection Tripped
	//36 SOP660_B1	AT %MX6.3	: BOOL;	// Conveyor Sensor
	//37 SOP670_FQ1	AT %MX6.4	: BOOL;	// Motor Protection Tripped
	//38 SOP670_B1	AT %MX6.5	: BOOL;	// Conveyor Sensor
	//39 SOP680_FQ1	AT %MX6.6	: BOOL;	// Motor Protection Tripped
	//40 SOP680_B1	AT %MX6.7	: BOOL;	// Conveyor Sensor
	//SOP004_A1_7_2	AT %MB7	: BYTE;	// 16 DI Card, Input 8-15 
	//Reserved	AT %MX7.0	: BOOL;	// 
	//Reserved	AT %MX7.1	: BOOL;	// 
	//Reserved	AT %MX7.2	: BOOL;	// 
	//Reserved	AT %MX7.3	: BOOL;	// 
	//Reserved	AT %MX7.4	: BOOL;	// 
	//Reserved	AT %MX7.5	: BOOL;	// 
	//Reserved	AT %MX7.6	: BOOL;	// 
	//Reserved	AT %MX7.7	: BOOL;	// 
	SOP004_A3_2	AT %MW4	: WORD;	// 16 DI Card, Input 0-7 
	//41 SOP690_S1	AT %MX8.0	: BOOL;	// Cycle Start
	//42 SOP690_S2	AT %MX8.1	: BOOL;	// Entry Request
	//43 SOP690_S3	AT %MX8.2	: BOOL;	// Reset Safety
	SOP690_NS1	AT %MX8.3	: BOOL;	// Emergency Stop
	//Reserved	AT %MX8.4	: BOOL;	// 
	//Reserved	AT %MX8.5	: BOOL;	// 
	//Reserved	AT %MX8.6	: BOOL;	// 
	//Reserved	AT %MX8.7	: BOOL;	// 
	//SOP004_A3_2_2	AT %MB9	: BYTE;	// 16 DI Card, Input 8-15 
	//44 SOP690_K1	AT %MX9.0	: BOOL;	// Gate Unlocked Confirmation
    //45 SOP690_B1	AT %MX9.1	: BOOL;	// Gate Closed
	//Reserved	AT %MX9.2	: BOOL;	// 
	//Reserved	AT %MX9.3	: BOOL;	// 
	//Reserved	AT %MX9.4	: BOOL;	// 
	//Reserved	AT %MX9.5	: BOOL;	// 
	//Reserved	AT %MX9.6	: BOOL;	// 
	//Reserved	AT %MX9.7	: BOOL;	// 

	(* OUTPUTS *)
	SOP004_A1_8	AT %QW0	: WORD;	// 16 DO Card, Output 0-7 
    //46 SOP040_K3	AT %QX0.0	: BOOL;	// Reset Safety circuit // Por declarar
	SOP040_K4	AT %QX0.1	: BOOL;	// Safety Power Line
	SOP040_K5	AT %QX0.2	: BOOL;	// Safety Pneumatics
	//Reserved	AT %QX0.3	: BOOL;	// 
	//Reserved	AT %QX0.4	: BOOL;	// 
	//47 SOP600_H1	AT %QX0.5	: BOOL;	// Control Voltage On Light
	//48 SOP600_H2	AT %QX0.6	: BOOL;	// Cycle Start Light
	//49 SOP600_H3	AT %QX0.7	: BOOL;	// Cycle Stop Light
	//SOP004_A1_8_2	AT %QB1	: BYTE;	// 16 DO Card, Output 8-15 
	//50 SOP600_H4	AT %QX1.0	: BOOL;	// Reset Alarm Light
	//51 SOP600_H5	AT %QX1.1	: BOOL;	// Reset Safety Light
	//52 SOP600_H6	AT %QX1.2	: BOOL;	// Blue Light
	//53 SOP600_H7	AT %QX1.3	: BOOL;	// Green Light
	//54 SOP600_H8	AT %QX1.4	: BOOL;	// Orange Light
	//55 SOP600_H9	AT %QX1.5	: BOOL;	// Red Light
	//56 SOP600_H10	AT %QX1.6	: BOOL;	// Home Position Light
	//57 SOP600_H11	AT %QX1.7	: BOOL;	// Horn sound
	SOP004_A1_9	AT %QW1	: WORD;	// 16 DO Card, Output 0-7 
	//58 SOP610_KM1	AT %QX2.0	: BOOL;	// Conveyor Forward
	//59 SOP610_KM2	AT %QX2.1	: BOOL;	// Conveyor Reverse
	//60 SOP620_KM1	AT %QX2.2	: BOOL;	// Conveyor Forward
	//61 SOP620_KM2	AT %QX2.3	: BOOL;	// Conveyor Reverse
	//62 SOP630_KM1	AT %QX2.4	: BOOL;	// Conveyor Forward
	//63 SOP630_KM2	AT %QX2.5	: BOOL;	// Conveyor Reverse
	//Reserved	AT %QX2.6	: BOOL;	// 
	//Reserved	AT %QX2.7	: BOOL;	// 
	//SOP004_A1_9_2	AT %QB3	: BYTE;	// 16 DO Card, Output 8-15 
	//64 SOP640_KM1	AT %QX3.0	: BOOL;	// Conveyor Forward
	//65 SOP640_KM2	AT %QX3.1	: BOOL;	// Conveyor Reverse
	//66 SOP640_Y1	AT %QX3.2	: BOOL;	// Front Clamp Up
	//67 SOP640_Y2	AT %QX3.3	: BOOL;	// Front Clamp Down
	//68 SOP640_Y3	AT %QX3.4	: BOOL;	// Rear Clamp Up
	//69 SOP640_Y4	AT %QX3.5	: BOOL;	// Rear Clamp Down
	//Reserved	AT %QX3.6	: BOOL;	// 
	//70 SOP640_K2	AT %QX3.7	: BOOL;	// Light Curtain Muting 
	SOP004_A1_10	AT %QW2	: WORD;	// 16 DO Card, Output 0-7 
	//71 SOP650_KM1	AT %QX4.0	: BOOL;	// Conveyor Forward
	//72 SOP650_KM2	AT %QX4.1	: BOOL;	// Conveyor Reverse
	//73 SOP660_KM1	AT %QX4.2	: BOOL;	// Conveyor Forward
	//74 SOP660_KM2	AT %QX4.3	: BOOL;	// Conveyor Reverse
	//75 SOP670_KM1	AT %QX4.4	: BOOL;	// Conveyor Forward
	//76 SOP670_KM2	AT %QX4.5	: BOOL;	// Conveyor Reverse
	//77 SOP680_KM1	AT %QX4.6	: BOOL;	// Conveyor Forward
	//78 SOP680_KM2	AT %QX4.7	: BOOL;	// Conveyor Reverse
	//SOP004_A1_10_2	AT %QB5	: BYTE;	// 16 DO Card, Output 8-15 
	//Reserved	AT %QX5.0	: BOOL;	// 
	//Reserved	AT %QX5.1	: BOOL;	// 
	//Reserved	AT %QX5.2	: BOOL;	// 
	//Reserved	AT %QX5.3	: BOOL;	// 
	//Reserved	AT %QX5.4	: BOOL;	// 
	//Reserved	AT %QX5.5	: BOOL;	// 
	//Reserved	AT %QX5.6	: BOOL;	// 
	//Reserved	AT %QX5.7	: BOOL;	// 
	SOP004_A3_3	AT %QW3	: WORD;	// 16 DO Card, Output 0-7 
	//79 SOP690_H1	AT %QX6.0	: BOOL;	// Cycle Start Light
	//80 SOP690_H2	AT %QX6.1	: BOOL;	// Entry Request Light
	//81 SOP690_H3	AT %QX6.2	: BOOL;	// Reset Safety Light
	//Reserved	AT %QX6.3	: BOOL;	// 
	//Reserved	AT %QX6.4	: BOOL;	// 
	//Reserved	AT %QX6.5	: BOOL;	// 
	//Reserved	AT %QX6.6	: BOOL;	// 
	//Reserved	AT %QX6.7	: BOOL;	// 
	//SOP004_A3_3_2	AT %QB7	: BYTE;	// 16 DO Card, Output 8-15 
	//82 SOP690_S4	AT %QX7.0	: BOOL;	// Unlock Gate
	//Reserved	AT %QX7.1	: BOOL;	// 
	//Reserved	AT %QX7.2	: BOOL;	// 
	//Reserved	AT %QX7.3	: BOOL;	// 
	//Reserved	AT %QX7.4	: BOOL;	// 
	//Reserved	AT %QX7.5	: BOOL;	// 
	//Reserved	AT %QX7.6	: BOOL;	// 
	//Reserved	AT %QX7.7	: BOOL;	// 	
END_VAR

// Device/Application/OP60_Main
PROGRAM OP60_Main
VAR
	
	RS_0: RS;
	Operator_Faulted: BOOL;
	RS_1: RS;
	Stop: BOOL;
END_VAR
VAR // added by the converter: edge detectors and wires of the graphical bodies
    _rt1, _rt2, _rt3 : R_TRIG;
    _w1, _w2, _w3, _w4 : BOOL;
    _ft1, _ft2 : F_TRIG;
END_VAR

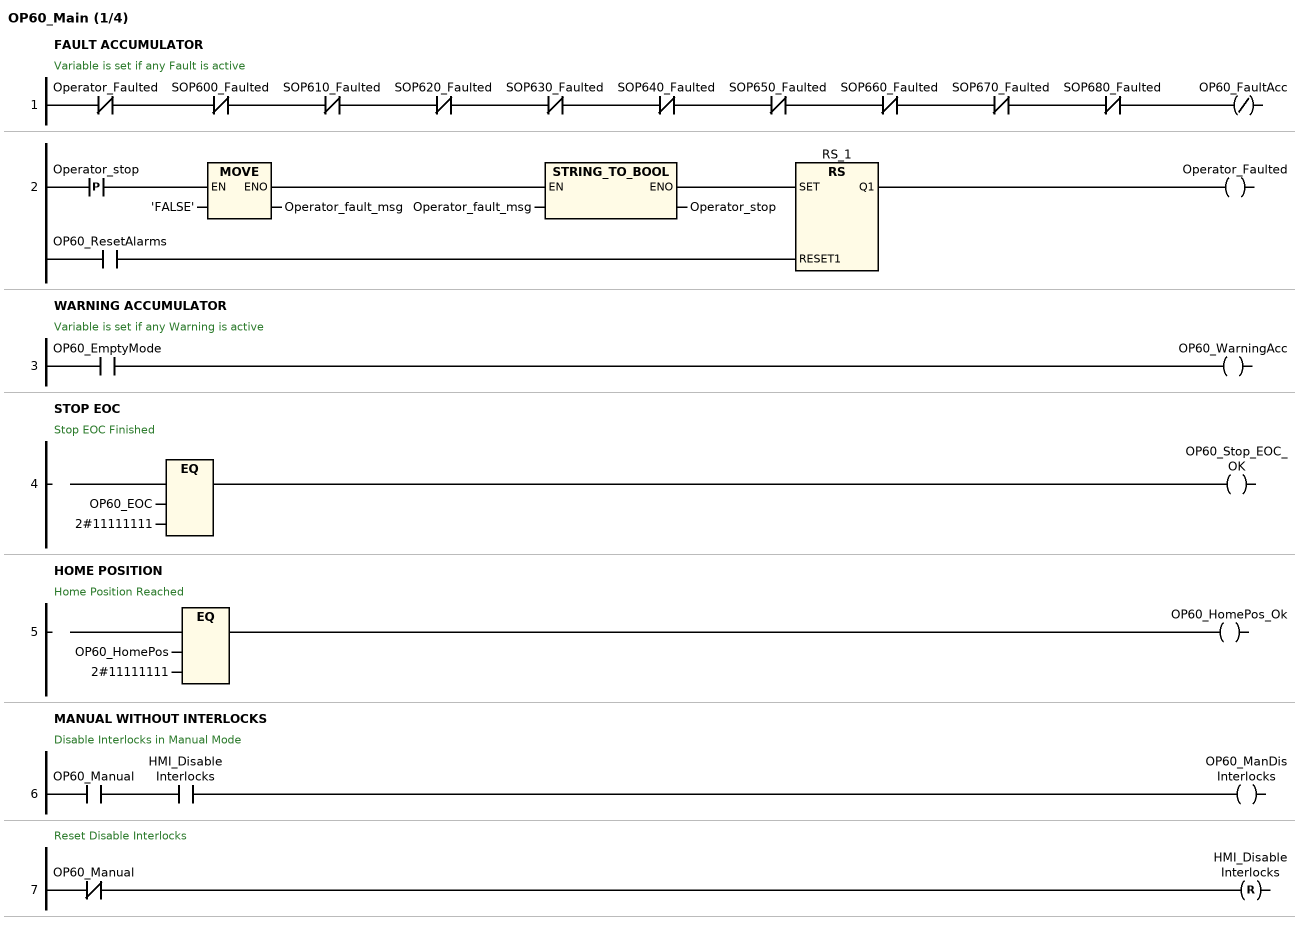
// NETWORK 1: FAULT ACCUMULATOR
// Variable is set if any Fault is active
OP60_FaultAcc := NOT (NOT Operator_Faulted AND NOT SOP600_Faulted AND NOT SOP610_Faulted AND NOT SOP620_Faulted AND NOT SOP630_Faulted AND NOT SOP640_Faulted AND NOT SOP650_Faulted AND NOT SOP660_Faulted AND NOT SOP670_Faulted AND NOT SOP680_Faulted);

// NETWORK 2
_rt1(CLK := Operator_stop);
_w1 := _rt1.Q;
IF _w1 THEN Operator_fault_msg := 'FALSE'; END_IF
IF _w1 THEN Operator_stop := STRING_TO_BOOL(Operator_fault_msg); END_IF
RS_1(SET := _w1, RESET1 := OP60_ResetAlarms); // RS
Operator_Faulted := RS_1.Q1;

// NETWORK 3: WARNING ACCUMULATOR
// Variable is set if any Warning is active
OP60_WarningAcc := OP60_EmptyMode;

// NETWORK 4: STOP EOC
// Stop EOC Finished
OP60_Stop_EOC_OK := OP60_EOC = 2#11111111;

// NETWORK 5: HOME POSITION
// Home Position Reached
OP60_HomePos_Ok := OP60_HomePos = 2#11111111;

// NETWORK 6: MANUAL WITHOUT INTERLOCKS
// Disable Interlocks in Manual Mode
OP60_ManDisInterlocks := OP60_Manual AND HMI_DisableInterlocks;

// NETWORK 7
// Reset Disable Interlocks
HMI_DisableInterlocks R= NOT OP60_Manual;

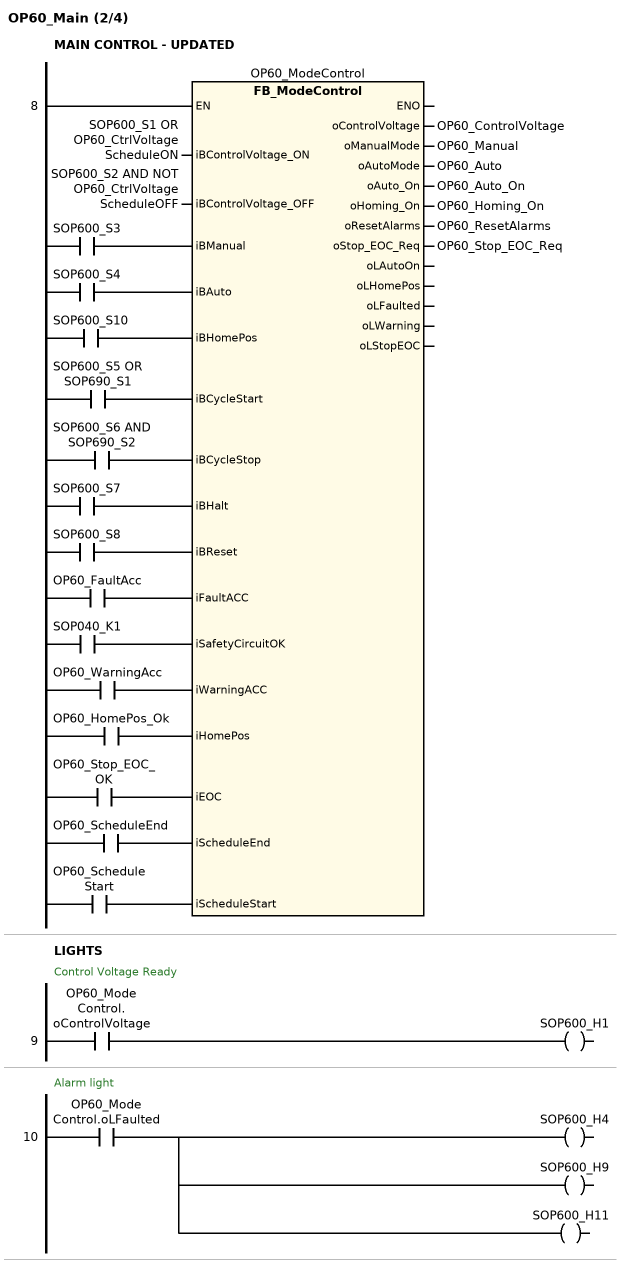
// NETWORK 8: MAIN CONTROL - UPDATED
OP60_ModeControl(
    iBControlVoltage_ON := SOP600_S1 OR OP60_CtrlVoltageScheduleON,
    iBControlVoltage_OFF := SOP600_S2 AND NOT OP60_CtrlVoltageScheduleOFF,
    iBManual := SOP600_S3,
    iBAuto := SOP600_S4,
    iBHomePos := SOP600_S10,
    iBCycleStart := SOP600_S5 OR SOP690_S1,
    iBCycleStop := SOP600_S6 AND SOP690_S2,
    iBHalt := SOP600_S7,
    iBReset := SOP600_S8,
    iFaultACC := OP60_FaultAcc,
    iSafetyCircuitOK := SOP040_K1,
    iWarningACC := OP60_WarningAcc,
    iHomePos := OP60_HomePos_Ok,
    iEOC := OP60_Stop_EOC_OK,
    iScheduleEnd := OP60_ScheduleEnd,
    iScheduleStart := OP60_ScheduleStart,
    oControlVoltage => OP60_ControlVoltage,
    oManualMode => OP60_Manual,
    oAutoMode => OP60_Auto,
    oAuto_On => OP60_Auto_On,
    oHoming_On => OP60_Homing_On,
    oResetAlarms => OP60_ResetAlarms,
    oStop_EOC_Req => OP60_Stop_EOC_Req); // FB_ModeControl

// NETWORK 9: LIGHTS
// Control Voltage Ready
SOP600_H1 := OP60_ModeControl.oControlVoltage;

// NETWORK 10
// Alarm light
SOP600_H4 := OP60_ModeControl.oLFaulted;
SOP600_H9 := OP60_ModeControl.oLFaulted;
SOP600_H11 := OP60_ModeControl.oLFaulted;

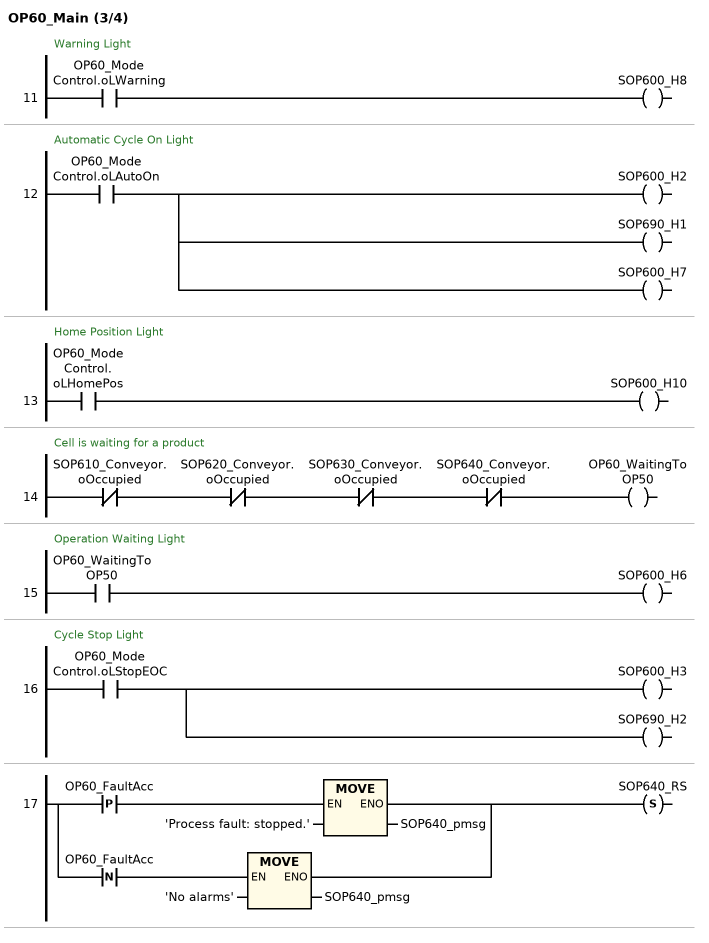
// NETWORK 11
// Warning Light
SOP600_H8 := OP60_ModeControl.oLWarning;

// NETWORK 12
// Automatic Cycle On Light
SOP600_H2 := OP60_ModeControl.oLAutoOn;
SOP690_H1 := OP60_ModeControl.oLAutoOn;
SOP600_H7 := OP60_ModeControl.oLAutoOn;

// NETWORK 13
// Home Position Light
SOP600_H10 := OP60_ModeControl.oLHomePos;

// NETWORK 14
// Cell is waiting for a product
OP60_WaitingToOP50 := NOT SOP610_Conveyor.oOccupied AND NOT SOP620_Conveyor.oOccupied AND NOT SOP630_Conveyor.oOccupied AND NOT SOP640_Conveyor.oOccupied;

// NETWORK 15
// Operation Waiting Light
SOP600_H6 := OP60_WaitingToOP50;

// NETWORK 16
// Cycle Stop Light
SOP600_H3 := OP60_ModeControl.oLStopEOC;
SOP690_H2 := OP60_ModeControl.oLStopEOC;

// NETWORK 17
_rt2(CLK := OP60_FaultAcc);
_w2 := _rt2.Q;
IF _w2 THEN SOP640_pmsg := 'Process fault: stopped.'; END_IF
_ft1(CLK := OP60_FaultAcc);
_w3 := _ft1.Q;
IF _w3 THEN SOP640_pmsg := 'No alarms'; END_IF
SOP640_RS S= _w2 OR _w3;

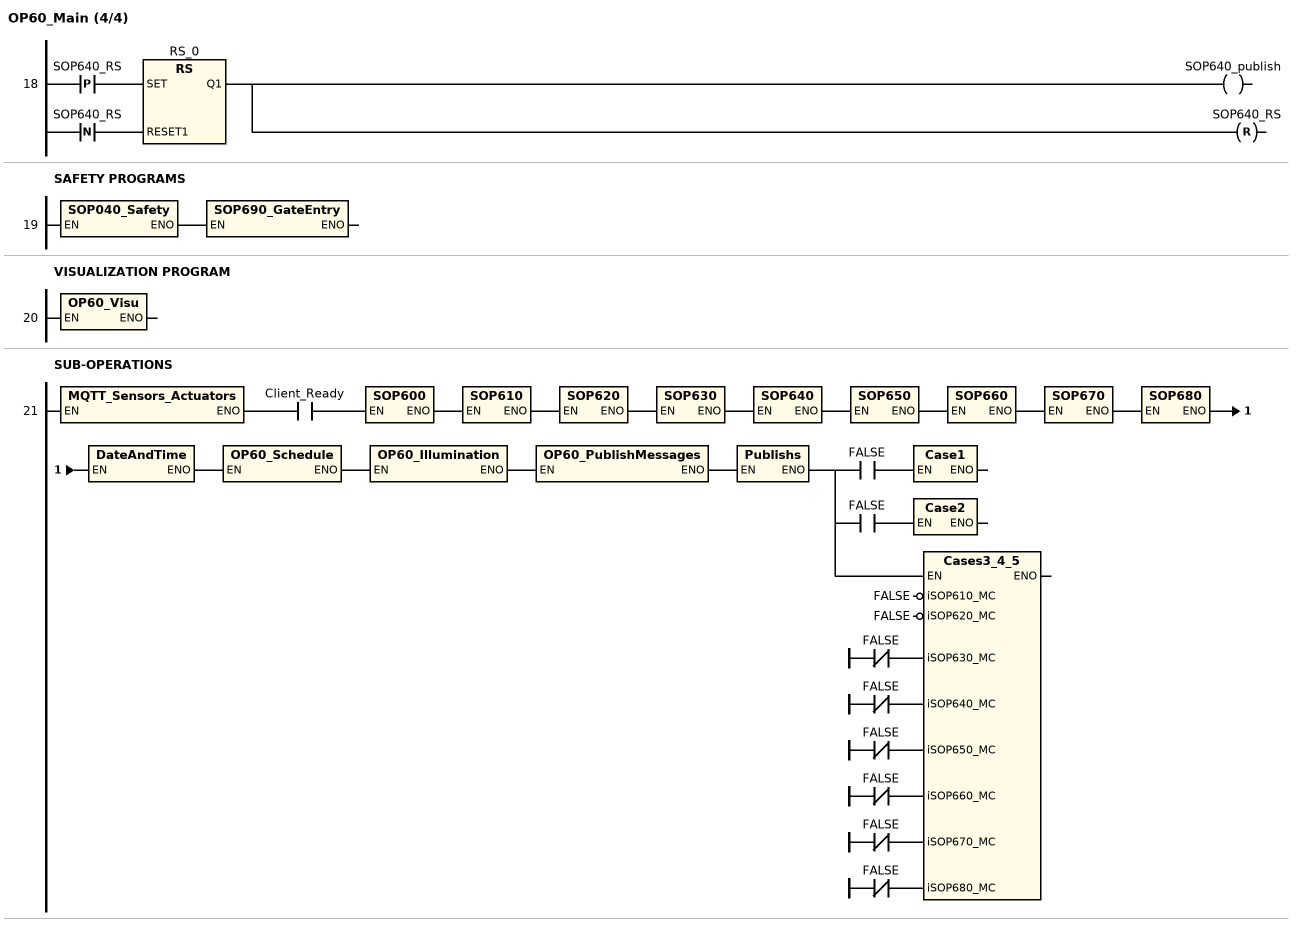
// NETWORK 18
_rt3(CLK := SOP640_RS);
_ft2(CLK := SOP640_RS);
RS_0(SET := _rt3.Q, RESET1 := _ft2.Q); // RS
SOP640_publish := RS_0.Q1;
SOP640_RS R= RS_0.Q1;

// NETWORK 19: SAFETY PROGRAMS
SOP040_Safety();
SOP690_GateEntry();

// NETWORK 20: VISUALIZATION PROGRAM
OP60_Visu();

// NETWORK 21: SUB-OPERATIONS
MQTT_Sensors_Actuators();
_w4 := Client_Ready;
IF _w4 THEN SOP600(); END_IF
IF _w4 THEN SOP610(); END_IF
IF _w4 THEN SOP620(); END_IF
IF _w4 THEN SOP630(); END_IF
IF _w4 THEN SOP640(); END_IF
IF _w4 THEN SOP650(); END_IF
IF _w4 THEN SOP660(); END_IF
IF _w4 THEN SOP670(); END_IF
IF _w4 THEN SOP680(); END_IF
IF _w4 THEN DateAndTime(); END_IF
IF _w4 THEN OP60_Schedule(); END_IF
IF _w4 THEN OP60_Illumination(); END_IF
IF _w4 THEN OP60_PublishMessages(); END_IF
IF _w4 THEN Publishs(); END_IF
IF _w4 AND FALSE THEN Case1(); END_IF
IF _w4 AND FALSE THEN Case2(); END_IF
IF _w4 THEN
    Cases3_4_5(iSOP610_MC := NOT FALSE, iSOP620_MC := NOT FALSE, iSOP630_MC := NOT FALSE, iSOP640_MC := NOT FALSE, iSOP650_MC := NOT FALSE, iSOP660_MC := NOT FALSE, iSOP670_MC := NOT FALSE, iSOP680_MC := NOT FALSE);
END_IF

END_PROGRAM

// Device/Application/FBs/FB_ModeControl
FUNCTION_BLOCK FB_ModeControl
VAR_INPUT
	iBControlVoltage_ON: BOOL; 		// Control Voltage On Button (NO)
	iBControlVoltage_OFF: BOOL; 	// Control Voltage Off Button (NC)
	iBManual: BOOL;					// Manual Mode Button (NO)
	iBAuto: BOOL;					// Automatic Mode Button (NO)
	iBHomePos: BOOL;				// Home Position Button (NO)
	iBCycleStart: BOOL;				// Cycle Start Button (NO)
	iBCycleStop: BOOL;				// Cycle Stop Button (NO)
	iBHalt: BOOL;					// Halt Button (NC)
	iBReset: BOOL;					// Reset Alarm Button (NO)
	iFaultACC: BOOL;				// Fault Accumulator
	iSafetyCircuitOK: BOOL;			// Safety Circuit OK
	iWarningACC: BOOL;				// Warning Accumulator
	iHomePos: BOOL;					// At Home Position
	iEOC: BOOL;						// End of Cycle Reached
	iScheduleEnd: BOOL;				// Schedule start
	iScheduleStart: BOOL;			// Schedule end
END_VAR
VAR_OUTPUT
	oControlVoltage: BOOL; 		// Control Voltage Ready
	oManualMode: BOOL;			// Manual Mode Active
	oAutoMode: BOOL;			// Automatic Mode Active
	oAuto_On: BOOL;				// Automatic Cycle On
	oHoming_On: BOOL;			// Homing Cycle On
	oResetAlarms: BOOL;			// Reset Alarms
	oStop_EOC_Req: BOOL;		// Stop EOC Requested
	oLAutoOn: BOOL;				// Automatic Cycle On Light 
	oLHomePos: BOOL;			// Home Position Light 
	oLFaulted: BOOL;			// Fault Light 
	oLWarning: BOOL;			// Warning Light 
	oLStopEOC: BOOL;			// Stop EOC Light 
END_VAR
VAR
	Timer_Auto_On: TON;
	Timer_Home_On: TON;
	Timer_Home2_On: TON;
	Timer1_Flash_1s: TON;
	Timer2_Flash_1s: TP;
	FaultAck: BOOL;				// Faults Acknowledge
	EOC_OK: BOOL;				// EOC Finished
	Homing_OK: BOOL;			// Homing Finished
	Home_Pos_Req: BOOL;			// Homing Requested
	CycleStartOK: BOOL;			// Cycle Start Conditions OK
END_VAR
VAR // added by the converter: edge detectors and wires of the graphical bodies
    _rt1, _rt2 : R_TRIG;
    _w1 : BOOL;
END_VAR

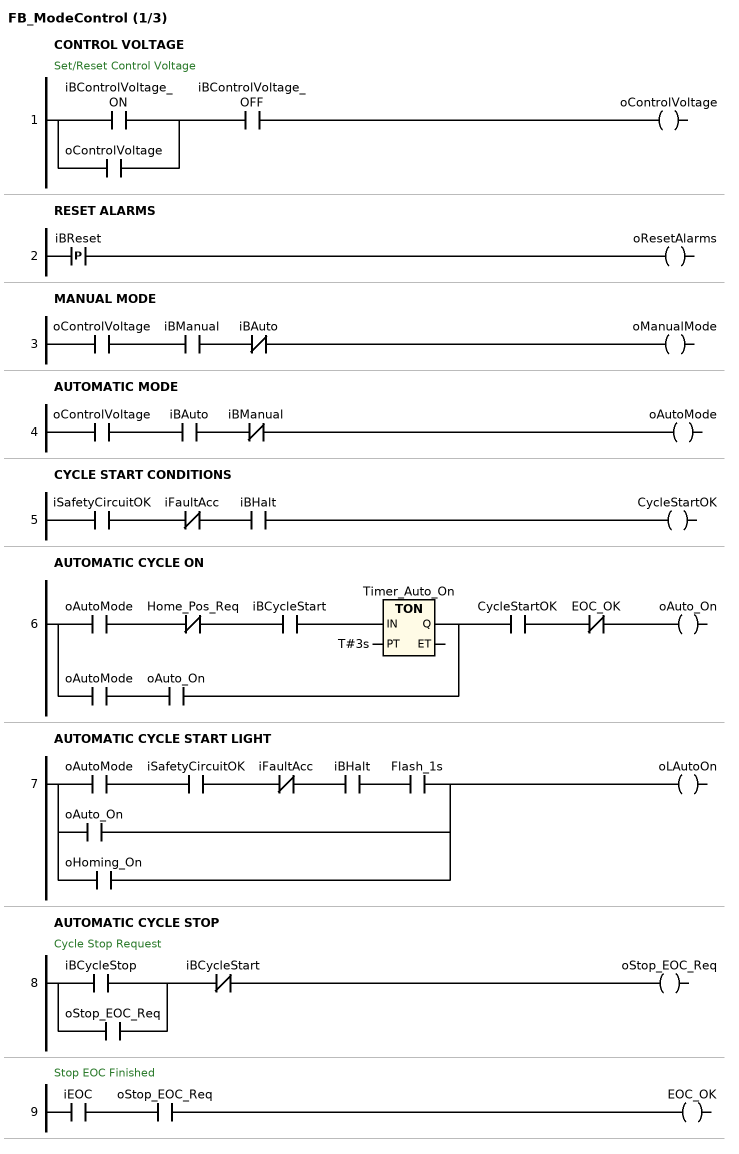
// NETWORK 1: CONTROL VOLTAGE
// Set/Reset Control Voltage
oControlVoltage := (iBControlVoltage_ON OR oControlVoltage) AND iBControlVoltage_OFF;

// NETWORK 2: RESET ALARMS
_rt1(CLK := iBReset);
oResetAlarms := _rt1.Q;

// NETWORK 3: MANUAL MODE
oManualMode := oControlVoltage AND iBManual AND NOT iBAuto;

// NETWORK 4: AUTOMATIC MODE
oAutoMode := oControlVoltage AND iBAuto AND NOT iBManual;

// NETWORK 5: CYCLE START CONDITIONS
CycleStartOK := iSafetyCircuitOK AND NOT iFaultAcc AND iBHalt;

// NETWORK 6: AUTOMATIC CYCLE ON
Timer_Auto_On(IN := oAutoMode AND NOT Home_Pos_Req AND iBCycleStart, PT := T#3s); // TON
oAuto_On := (Timer_Auto_On.Q OR oAutoMode AND oAuto_On) AND CycleStartOK AND NOT EOC_OK;

// NETWORK 7: AUTOMATIC CYCLE START LIGHT
oLAutoOn := oAutoMode AND iSafetyCircuitOK AND NOT iFaultAcc AND iBHalt AND Flash_1s OR oAuto_On OR oHoming_On;

// NETWORK 8: AUTOMATIC CYCLE STOP
// Cycle Stop Request
oStop_EOC_Req := (iBCycleStop OR oStop_EOC_Req) AND NOT iBCycleStart;

// NETWORK 9
// Stop EOC Finished
EOC_OK := iEOC AND oStop_EOC_Req;

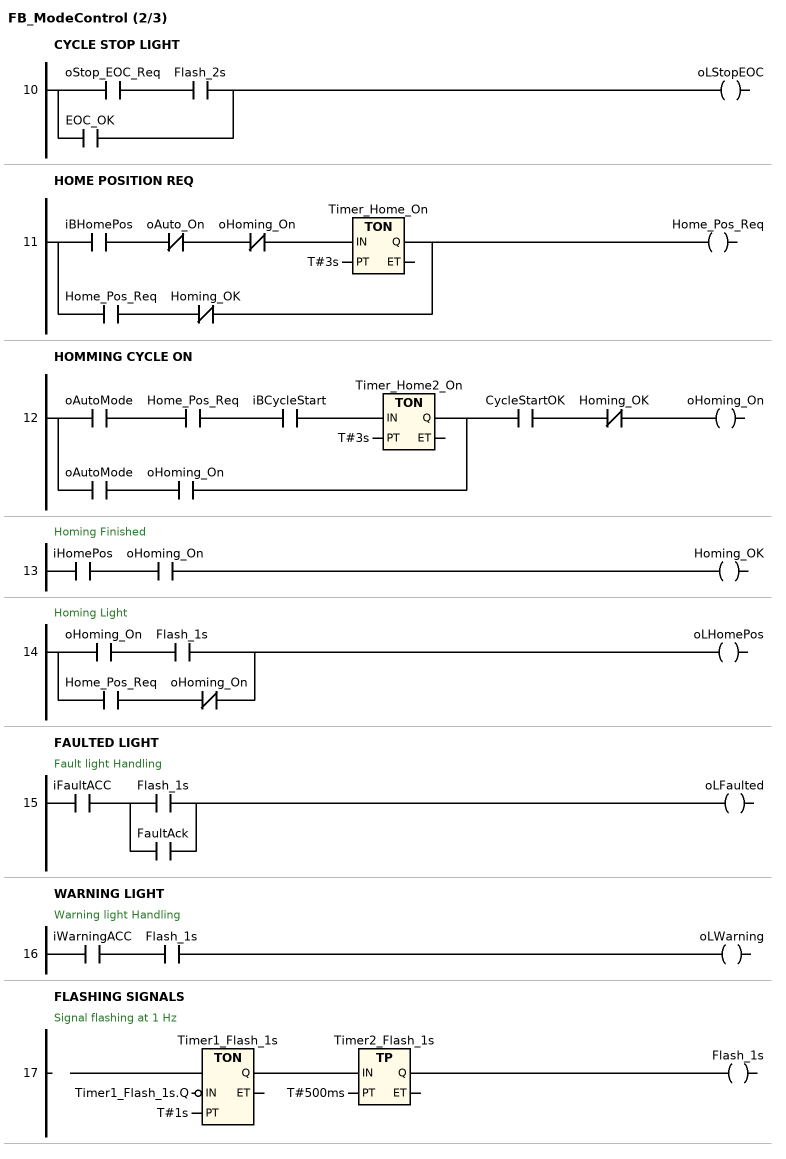
// NETWORK 10: CYCLE STOP LIGHT
oLStopEOC := oStop_EOC_Req AND Flash_2s OR EOC_OK;

// NETWORK 11: HOME POSITION REQ
Timer_Home_On(IN := iBHomePos AND NOT oAuto_On AND NOT oHoming_On, PT := T#3s); // TON
Home_Pos_Req := Timer_Home_On.Q OR Home_Pos_Req AND NOT Homing_OK;

// NETWORK 12: HOMMING CYCLE ON
Timer_Home2_On(IN := oAutoMode AND Home_Pos_Req AND iBCycleStart, PT := T#3s); // TON
oHoming_On := (Timer_Home2_On.Q OR oAutoMode AND oHoming_On) AND CycleStartOK AND NOT Homing_OK;

// NETWORK 13
// Homing Finished
Homing_OK := iHomePos AND oHoming_On;

// NETWORK 14
// Homing Light
oLHomePos := oHoming_On AND Flash_1s OR Home_Pos_Req AND NOT oHoming_On;

// NETWORK 15: FAULTED LIGHT
// Fault light Handling
oLFaulted := iFaultACC AND (Flash_1s OR FaultAck);

// NETWORK 16: WARNING LIGHT
// Warning light Handling
oLWarning := iWarningACC AND Flash_1s;

// NETWORK 17: FLASHING SIGNALS
// Signal flashing at 1 Hz
Timer1_Flash_1s(IN := NOT Timer1_Flash_1s.Q, PT := T#1s); // TON
Timer2_Flash_1s(IN := Timer1_Flash_1s.Q, PT := T#500ms); // TP
Flash_1s := Timer2_Flash_1s.Q;

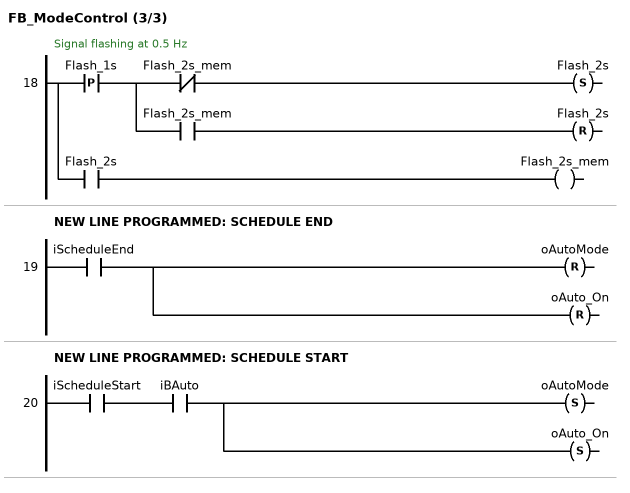
// NETWORK 18
// Signal flashing at 0.5 Hz
_rt2(CLK := Flash_1s);
Flash_2s S= _rt2.Q AND NOT Flash_2s_mem;
Flash_2s R= _rt2.Q AND Flash_2s_mem;
Flash_2s_mem := Flash_2s;

// NETWORK 19: NEW LINE PROGRAMMED: SCHEDULE END
oAutoMode R= iScheduleEnd;
oAuto_On R= iScheduleEnd;

// NETWORK 20: NEW LINE PROGRAMMED: SCHEDULE START
_w1 := iScheduleStart AND iBAuto;
oAutoMode S= _w1;
oAuto_On S= _w1;

END_FUNCTION_BLOCK

// Device/Application/SOP690_GateEntry
PROGRAM SOP690_GateEntry
VAR
	SOP690_RFID_Correct: BOOL;
	Prueba: BOOL;
	Prueba2: BOOL;
	Trigger: BOOL;
END_VAR
VAR // added by the converter: edge detectors and wires of the graphical bodies
    _ft1 : F_TRIG;
    _w1 : BOOL;
END_VAR

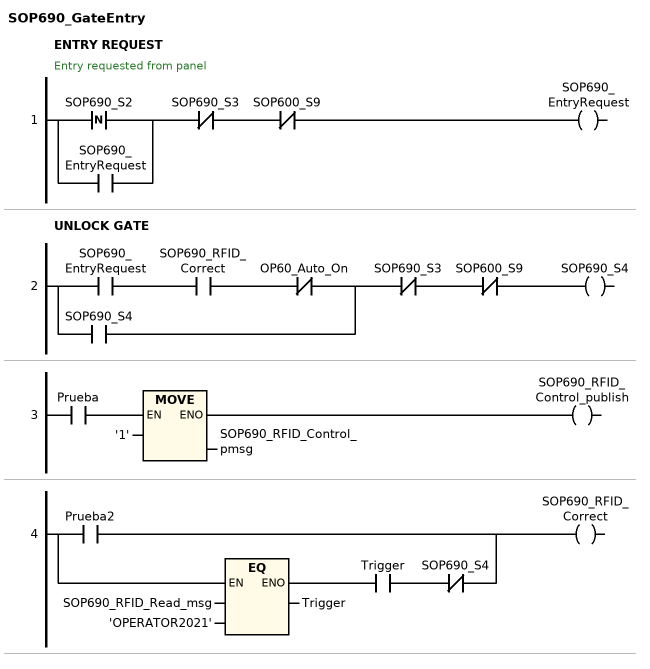
// NETWORK 1: ENTRY REQUEST
// Entry requested from panel
_ft1(CLK := SOP690_S2);
SOP690_EntryRequest := (_ft1.Q OR SOP690_EntryRequest) AND NOT SOP690_S3 AND NOT SOP600_S9;

// NETWORK 2: UNLOCK GATE
SOP690_S4 := (SOP690_EntryRequest AND SOP690_RFID_Correct AND NOT OP60_Auto_On OR SOP690_S4) AND NOT SOP690_S3 AND NOT SOP600_S9;

// NETWORK 3
_w1 := Prueba;
IF _w1 THEN SOP690_RFID_Control_pmsg := '1'; END_IF
SOP690_RFID_Control_publish := _w1;

// NETWORK 4
Trigger := SOP690_RFID_Read_msg = 'OPERATOR2021';
SOP690_RFID_Correct := Prueba2 OR Trigger AND NOT SOP690_S4;

END_PROGRAM

// Device/Application/SOP040_Safety
PROGRAM SOP040_Safety
VAR
END_VAR
VAR // added by the converter: edge detectors and wires of the graphical bodies
    _w1, _w2 : BOOL;
END_VAR

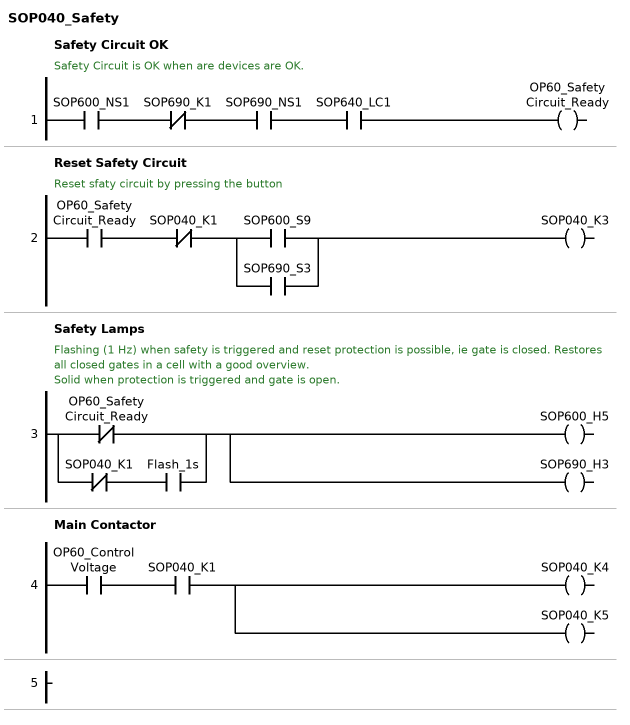
// NETWORK 1: Safety Circuit OK
// Safety Circuit is OK when are devices are OK.
OP60_SafetyCircuit_Ready := SOP600_NS1 AND NOT SOP690_K1 AND SOP690_NS1 AND SOP640_LC1;

// NETWORK 2: Reset Safety Circuit
// Reset sfaty circuit by pressing the button
SOP040_K3 := OP60_SafetyCircuit_Ready AND NOT SOP040_K1 AND (SOP600_S9 OR SOP690_S3);

// NETWORK 3: Safety Lamps
// Flashing (1 Hz) when safety is triggered and reset protection is possible, ie gate is closed. Restores all closed gates in a cell with a good overview.
// Solid when protection is triggered and gate is open.
_w1 := NOT OP60_SafetyCircuit_Ready OR NOT SOP040_K1 AND Flash_1s;
SOP600_H5 := _w1;
SOP690_H3 := _w1;

// NETWORK 4: Main Contactor
_w2 := OP60_ControlVoltage AND SOP040_K1;
SOP040_K4 := _w2;
SOP040_K5 := _w2;

// NETWORK 5

END_PROGRAM

// Device/Application/OP60_Visu
PROGRAM OP60_Visu
VAR
	CV_Overview: BOOL;
	CV_Process: BOOL;
	CV_Manual_SOP610t630: BOOL;
	CV_Manual_SOP640: BOOL;
	CV_Manual_SOP650t680: BOOL;
	CV_Production: BOOL;
	CV_Diagnostics: BOOL;
	CV_Interfaces: BOOL;
END_VAR

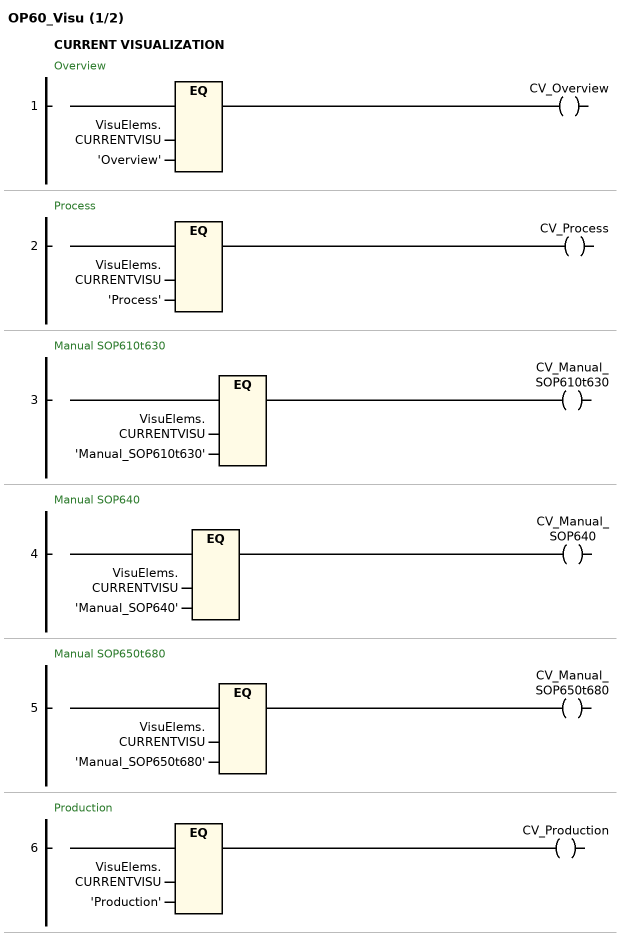
// NETWORK 1: CURRENT VISUALIZATION
// Overview
CV_Overview := VisuElems.CURRENTVISU = 'Overview';

// NETWORK 2
// Process
CV_Process := VisuElems.CURRENTVISU = 'Process';

// NETWORK 3
// Manual SOP610t630
CV_Manual_SOP610t630 := VisuElems.CURRENTVISU = 'Manual_SOP610t630';

// NETWORK 4
// Manual SOP640
CV_Manual_SOP640 := VisuElems.CURRENTVISU = 'Manual_SOP640';

// NETWORK 5
// Manual SOP650t680
CV_Manual_SOP650t680 := VisuElems.CURRENTVISU = 'Manual_SOP650t680';

// NETWORK 6
// Production
CV_Production := VisuElems.CURRENTVISU = 'Production';

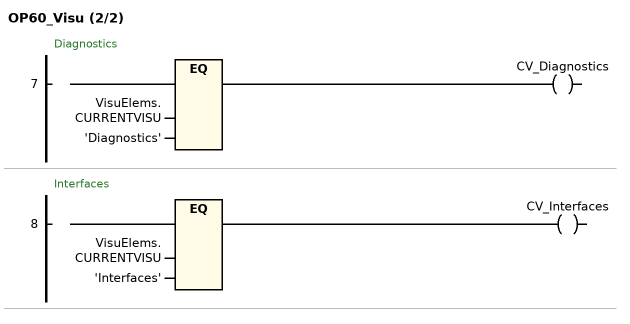
// NETWORK 7
// Diagnostics
CV_Diagnostics := VisuElems.CURRENTVISU = 'Diagnostics';

// NETWORK 8
// Interfaces
CV_Interfaces := VisuElems.CURRENTVISU = 'Interfaces';

END_PROGRAM

// Device/Application/OP60_PublishMessages
PROGRAM OP60_PublishMessages
VAR
	
	Initiate: BOOL := TRUE;
	SOP620_KM1_2_last_pmsg: STRING(1024);
	Trigger: BOOL;
	SOP610_KM1_2_last_pmsg: STRING(1024);
	SOP630_KM1_2_last_pmsg: STRING(1024);
	SOP640_KM1_2_last_pmsg: STRING(1024);
	SOP650_KM1_2_last_pmsg: STRING(1024);
	SOP660_KM1_2_last_pmsg: STRING(1024);
	SOP670_KM1_2_last_pmsg: STRING(1024);
	SOP680_KM1_2_last_pmsg: STRING(1024);
	SOP010_K3: BOOL;
END_VAR
VAR // added by the converter: edge detectors and wires of the graphical bodies
    _rt1, _rt2, _rt3, _rt4, _rt5, _rt6, _rt7, _rt8, _rt9, _rt10, _rt11, _rt12, _rt13, _rt14, _rt15, _rt16, _rt17, _rt18, _rt19, _rt20, _rt21, _rt22, _rt23, _rt24, _rt25, _rt26, _rt27, _rt28, _rt29, _rt30, _rt31, _rt32, _rt33, _rt34, _rt35, _rt36, _rt37, _rt38, _rt39, _rt40, _rt41, _rt42, _rt43, _rt44, _rt45, _rt46, _rt47, _rt48, _rt49, _rt50, _rt51, _rt52, _rt53, _rt54, _rt55, _rt56, _rt57, _rt58, _rt59, _rt60, _rt61, _rt62, _rt63, _rt64 : R_TRIG;
    _w1, _w2, _w3, _w4, _w5, _w6, _w7, _w8, _w9, _w10, _w11, _w12, _w13, _w14, _w15, _w16, _w17, _w18, _w19, _w20, _w21, _w22, _w23, _w24, _w25, _w26, _w27, _w28, _w29, _w30, _w31, _w32, _w33, _w34, _w35, _w36, _w37, _w38, _w39, _w40, _w41, _w42, _w43, _w44, _w45, _w46, _w47, _w48, _w49, _w50, _w51, _w52, _w53, _w54, _w55, _w56, _w57, _w58, _w59, _w60, _w61, _w62, _w63, _w64, _w65, _w66, _w67, _w68, _w69, _w70, _w71, _w72, _w73, _w74, _w75, _w76 : BOOL;
    _ft1, _ft2, _ft3, _ft4, _ft5, _ft6, _ft7, _ft8, _ft9, _ft10, _ft11, _ft12, _ft13, _ft14, _ft15, _ft16, _ft17, _ft18, _ft19, _ft20, _ft21, _ft22, _ft23, _ft24, _ft25, _ft26, _ft27, _ft28, _ft29, _ft30, _ft31, _ft32, _ft33, _ft34, _ft35, _ft36, _ft37 : F_TRIG;
END_VAR

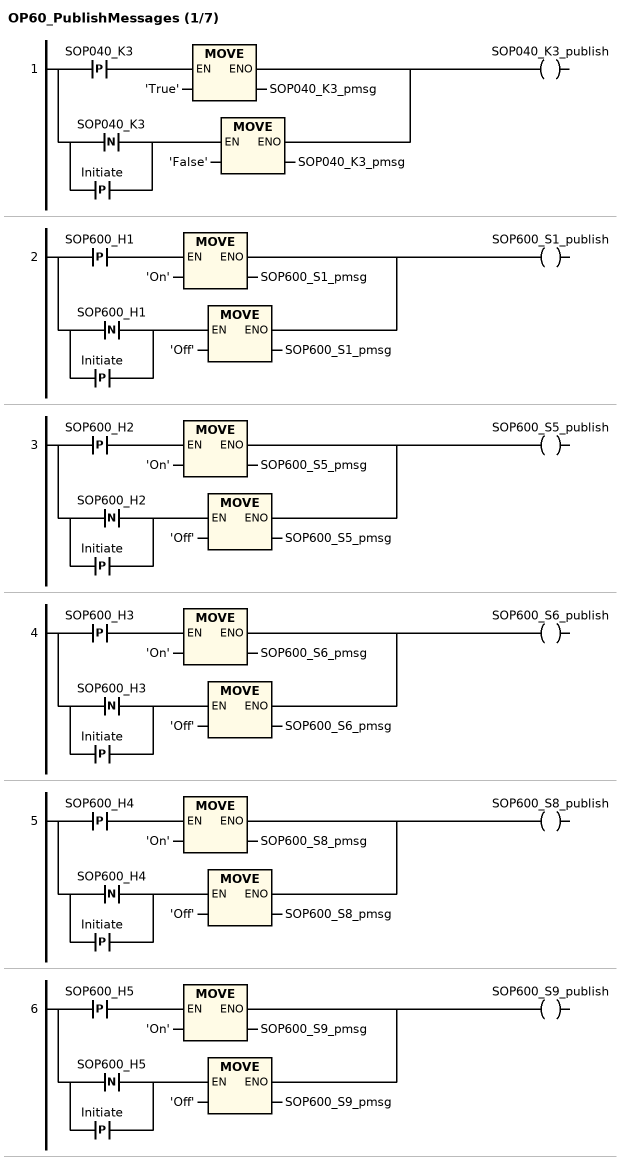
// NETWORK 1
_rt1(CLK := SOP040_K3);
_w1 := _rt1.Q;
IF _w1 THEN SOP040_K3_pmsg := 'True'; END_IF
_ft1(CLK := SOP040_K3);
_rt2(CLK := Initiate);
_w2 := _ft1.Q OR _rt2.Q;
IF _w2 THEN SOP040_K3_pmsg := 'False'; END_IF
SOP040_K3_publish := _w1 OR _w2;

// NETWORK 2
_rt3(CLK := SOP600_H1);
_w3 := _rt3.Q;
IF _w3 THEN SOP600_S1_pmsg := 'On'; END_IF
_ft2(CLK := SOP600_H1);
_rt4(CLK := Initiate);
_w4 := _ft2.Q OR _rt4.Q;
IF _w4 THEN SOP600_S1_pmsg := 'Off'; END_IF
SOP600_S1_publish := _w3 OR _w4;

// NETWORK 3
_rt5(CLK := SOP600_H2);
_w5 := _rt5.Q;
IF _w5 THEN SOP600_S5_pmsg := 'On'; END_IF
_ft3(CLK := SOP600_H2);
_rt6(CLK := Initiate);
_w6 := _ft3.Q OR _rt6.Q;
IF _w6 THEN SOP600_S5_pmsg := 'Off'; END_IF
SOP600_S5_publish := _w5 OR _w6;

// NETWORK 4
_rt7(CLK := SOP600_H3);
_w7 := _rt7.Q;
IF _w7 THEN SOP600_S6_pmsg := 'On'; END_IF
_ft4(CLK := SOP600_H3);
_rt8(CLK := Initiate);
_w8 := _ft4.Q OR _rt8.Q;
IF _w8 THEN SOP600_S6_pmsg := 'Off'; END_IF
SOP600_S6_publish := _w7 OR _w8;

// NETWORK 5
_rt9(CLK := SOP600_H4);
_w9 := _rt9.Q;
IF _w9 THEN SOP600_S8_pmsg := 'On'; END_IF
_ft5(CLK := SOP600_H4);
_rt10(CLK := Initiate);
_w10 := _ft5.Q OR _rt10.Q;
IF _w10 THEN SOP600_S8_pmsg := 'Off'; END_IF
SOP600_S8_publish := _w9 OR _w10;

// NETWORK 6
_rt11(CLK := SOP600_H5);
_w11 := _rt11.Q;
IF _w11 THEN SOP600_S9_pmsg := 'On'; END_IF
_ft6(CLK := SOP600_H5);
_rt12(CLK := Initiate);
_w12 := _ft6.Q OR _rt12.Q;
IF _w12 THEN SOP600_S9_pmsg := 'Off'; END_IF
SOP600_S9_publish := _w11 OR _w12;

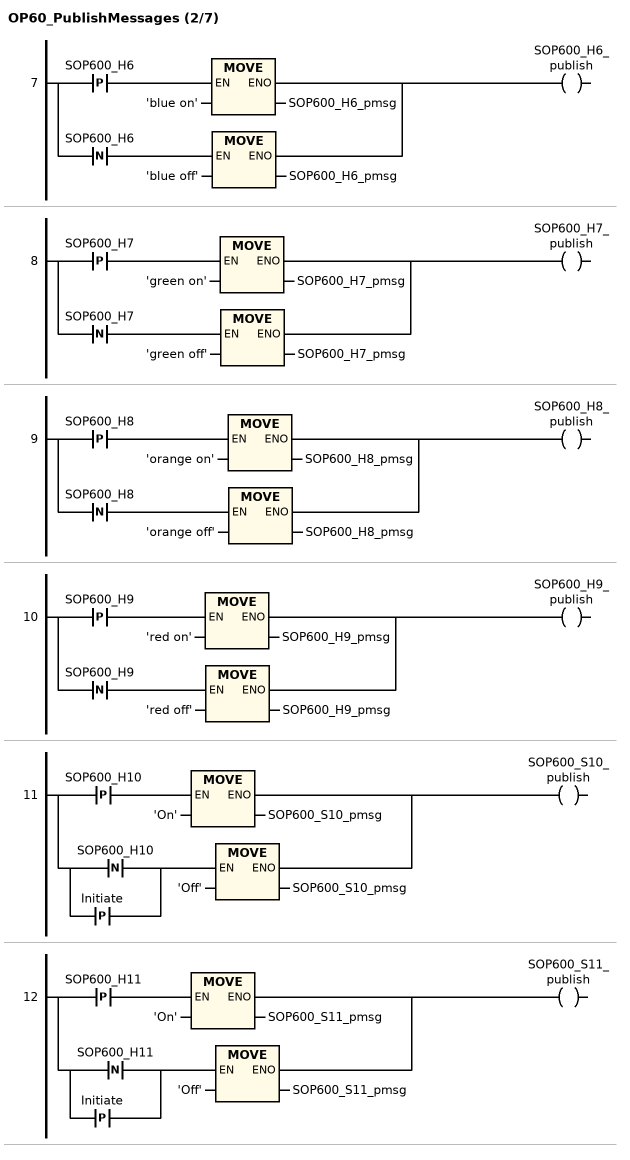
// NETWORK 7
_rt13(CLK := SOP600_H6);
_w13 := _rt13.Q;
IF _w13 THEN SOP600_H6_pmsg := 'blue on'; END_IF
_ft7(CLK := SOP600_H6);
_w14 := _ft7.Q;
IF _w14 THEN SOP600_H6_pmsg := 'blue off'; END_IF
SOP600_H6_publish := _w13 OR _w14;

// NETWORK 8
_rt14(CLK := SOP600_H7);
_w15 := _rt14.Q;
IF _w15 THEN SOP600_H7_pmsg := 'green on'; END_IF
_ft8(CLK := SOP600_H7);
_w16 := _ft8.Q;
IF _w16 THEN SOP600_H7_pmsg := 'green off'; END_IF
SOP600_H7_publish := _w15 OR _w16;

// NETWORK 9
_rt15(CLK := SOP600_H8);
_w17 := _rt15.Q;
IF _w17 THEN SOP600_H8_pmsg := 'orange on'; END_IF
_ft9(CLK := SOP600_H8);
_w18 := _ft9.Q;
IF _w18 THEN SOP600_H8_pmsg := 'orange off'; END_IF
SOP600_H8_publish := _w17 OR _w18;

// NETWORK 10
_rt16(CLK := SOP600_H9);
_w19 := _rt16.Q;
IF _w19 THEN SOP600_H9_pmsg := 'red on'; END_IF
_ft10(CLK := SOP600_H9);
_w20 := _ft10.Q;
IF _w20 THEN SOP600_H9_pmsg := 'red off'; END_IF
SOP600_H9_publish := _w19 OR _w20;

// NETWORK 11
_rt17(CLK := SOP600_H10);
_w21 := _rt17.Q;
IF _w21 THEN SOP600_S10_pmsg := 'On'; END_IF
_ft11(CLK := SOP600_H10);
_rt18(CLK := Initiate);
_w22 := _ft11.Q OR _rt18.Q;
IF _w22 THEN SOP600_S10_pmsg := 'Off'; END_IF
SOP600_S10_publish := _w21 OR _w22;

// NETWORK 12
_rt19(CLK := SOP600_H11);
_w23 := _rt19.Q;
IF _w23 THEN SOP600_S11_pmsg := 'On'; END_IF
_ft12(CLK := SOP600_H11);
_rt20(CLK := Initiate);
_w24 := _ft12.Q OR _rt20.Q;
IF _w24 THEN SOP600_S11_pmsg := 'Off'; END_IF
SOP600_S11_publish := _w23 OR _w24;

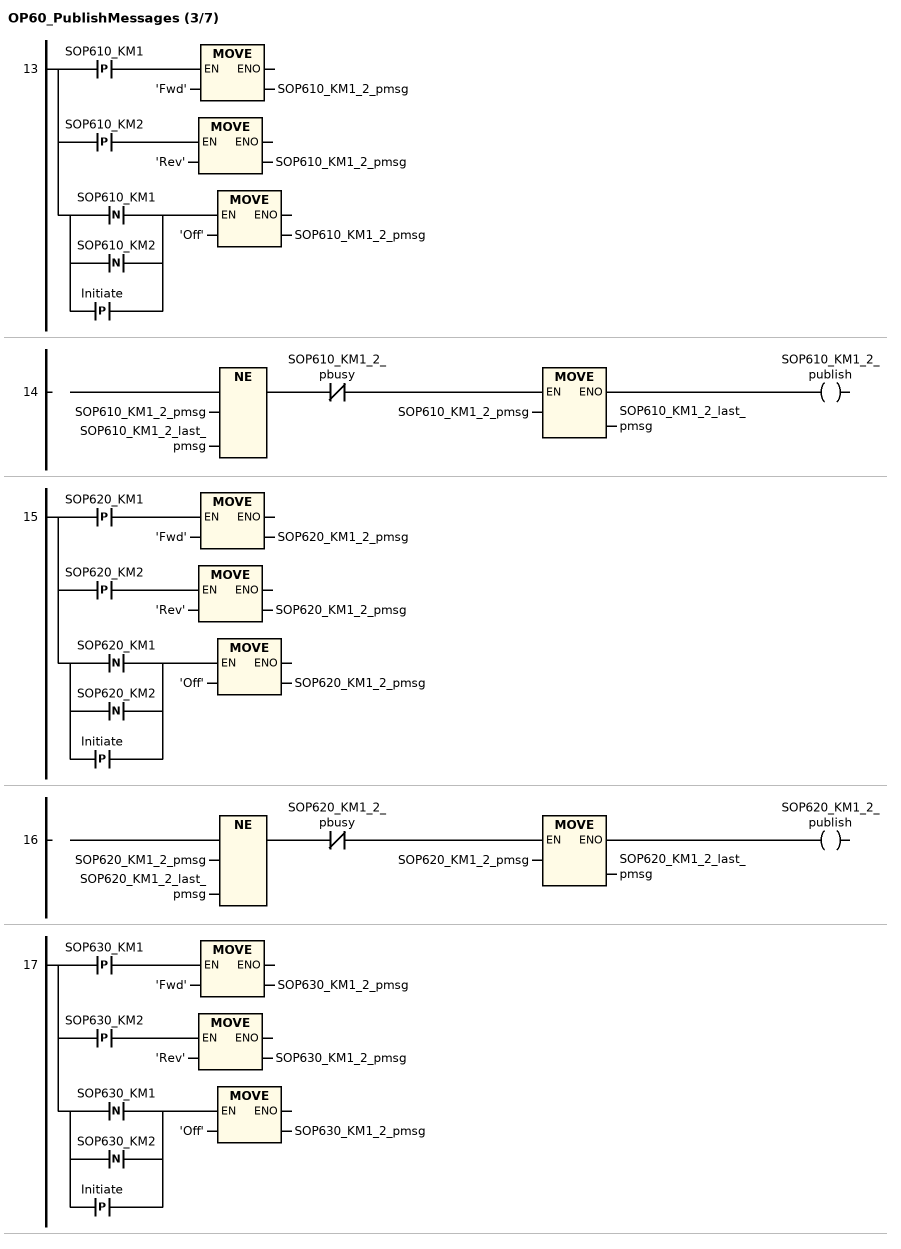
// NETWORK 13
_rt21(CLK := SOP610_KM1);
_w25 := _rt21.Q;
IF _w25 THEN SOP610_KM1_2_pmsg := 'Fwd'; END_IF
_rt22(CLK := SOP610_KM2);
_w26 := _rt22.Q;
IF _w26 THEN SOP610_KM1_2_pmsg := 'Rev'; END_IF
_ft13(CLK := SOP610_KM1);
_ft14(CLK := SOP610_KM2);
_rt23(CLK := Initiate);
_w27 := _ft13.Q OR _ft14.Q OR _rt23.Q;
IF _w27 THEN SOP610_KM1_2_pmsg := 'Off'; END_IF
(* _w25 OR _w26 OR _w27; result not used *)

// NETWORK 14
_w28 := SOP610_KM1_2_pmsg <> SOP610_KM1_2_last_pmsg AND NOT SOP610_KM1_2_pbusy;
IF _w28 THEN SOP610_KM1_2_last_pmsg := SOP610_KM1_2_pmsg; END_IF
SOP610_KM1_2_publish := _w28;

// NETWORK 15
_rt24(CLK := SOP620_KM1);
_w29 := _rt24.Q;
IF _w29 THEN SOP620_KM1_2_pmsg := 'Fwd'; END_IF
_rt25(CLK := SOP620_KM2);
_w30 := _rt25.Q;
IF _w30 THEN SOP620_KM1_2_pmsg := 'Rev'; END_IF
_ft15(CLK := SOP620_KM1);
_ft16(CLK := SOP620_KM2);
_rt26(CLK := Initiate);
_w31 := _ft15.Q OR _ft16.Q OR _rt26.Q;
IF _w31 THEN SOP620_KM1_2_pmsg := 'Off'; END_IF
(* _w29 OR _w30 OR _w31; result not used *)

// NETWORK 16
_w32 := SOP620_KM1_2_pmsg <> SOP620_KM1_2_last_pmsg AND NOT SOP620_KM1_2_pbusy;
IF _w32 THEN SOP620_KM1_2_last_pmsg := SOP620_KM1_2_pmsg; END_IF
SOP620_KM1_2_publish := _w32;

// NETWORK 17
_rt27(CLK := SOP630_KM1);
_w33 := _rt27.Q;
IF _w33 THEN SOP630_KM1_2_pmsg := 'Fwd'; END_IF
_rt28(CLK := SOP630_KM2);
_w34 := _rt28.Q;
IF _w34 THEN SOP630_KM1_2_pmsg := 'Rev'; END_IF
_ft17(CLK := SOP630_KM1);
_ft18(CLK := SOP630_KM2);
_rt29(CLK := Initiate);
_w35 := _ft17.Q OR _ft18.Q OR _rt29.Q;
IF _w35 THEN SOP630_KM1_2_pmsg := 'Off'; END_IF
(* _w33 OR _w34 OR _w35; result not used *)

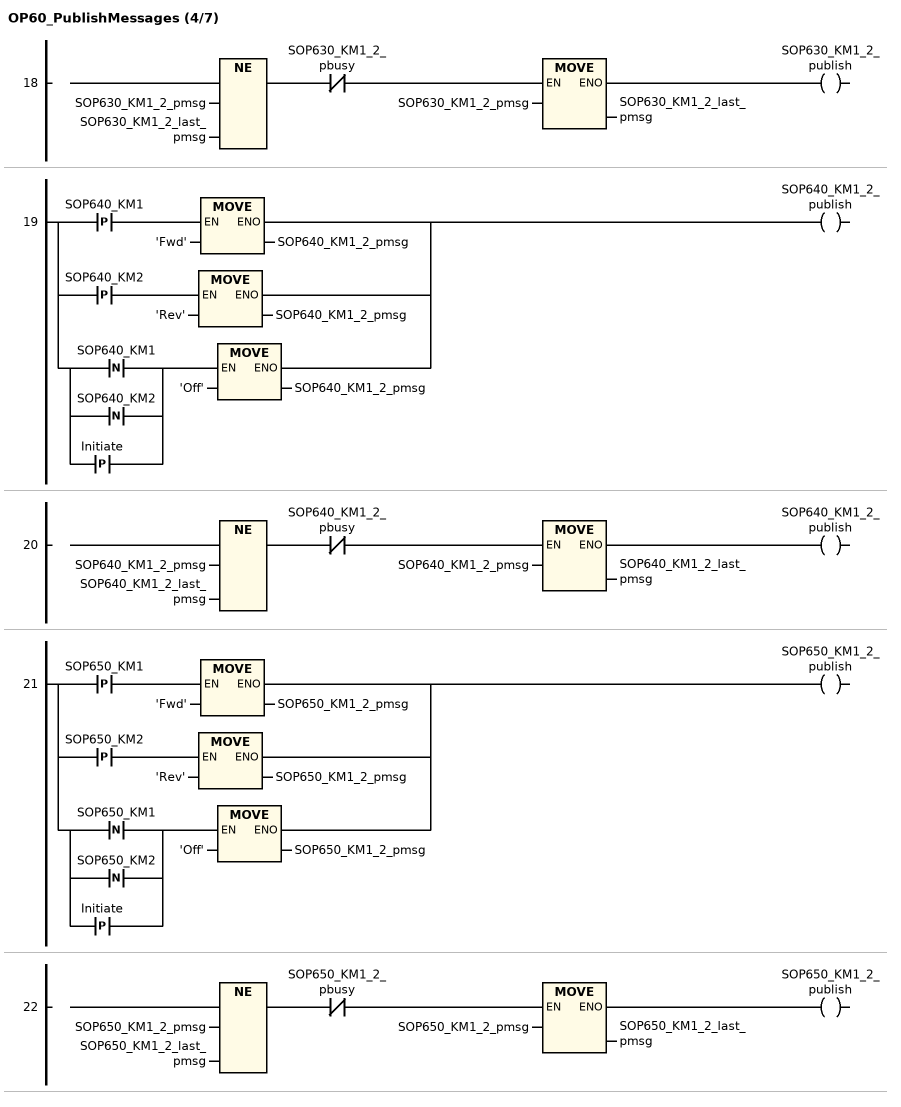
// NETWORK 18
_w36 := SOP630_KM1_2_pmsg <> SOP630_KM1_2_last_pmsg AND NOT SOP630_KM1_2_pbusy;
IF _w36 THEN SOP630_KM1_2_last_pmsg := SOP630_KM1_2_pmsg; END_IF
SOP630_KM1_2_publish := _w36;

// NETWORK 19
_rt30(CLK := SOP640_KM1);
_w37 := _rt30.Q;
IF _w37 THEN SOP640_KM1_2_pmsg := 'Fwd'; END_IF
_rt31(CLK := SOP640_KM2);
_w38 := _rt31.Q;
IF _w38 THEN SOP640_KM1_2_pmsg := 'Rev'; END_IF
_ft19(CLK := SOP640_KM1);
_ft20(CLK := SOP640_KM2);
_rt32(CLK := Initiate);
_w39 := _ft19.Q OR _ft20.Q OR _rt32.Q;
IF _w39 THEN SOP640_KM1_2_pmsg := 'Off'; END_IF
SOP640_KM1_2_publish := _w37 OR _w38 OR _w39;

// NETWORK 20
_w40 := SOP640_KM1_2_pmsg <> SOP640_KM1_2_last_pmsg AND NOT SOP640_KM1_2_pbusy;
IF _w40 THEN SOP640_KM1_2_last_pmsg := SOP640_KM1_2_pmsg; END_IF
SOP640_KM1_2_publish := _w40;

// NETWORK 21
_rt33(CLK := SOP650_KM1);
_w41 := _rt33.Q;
IF _w41 THEN SOP650_KM1_2_pmsg := 'Fwd'; END_IF
_rt34(CLK := SOP650_KM2);
_w42 := _rt34.Q;
IF _w42 THEN SOP650_KM1_2_pmsg := 'Rev'; END_IF
_ft21(CLK := SOP650_KM1);
_ft22(CLK := SOP650_KM2);
_rt35(CLK := Initiate);
_w43 := _ft21.Q OR _ft22.Q OR _rt35.Q;
IF _w43 THEN SOP650_KM1_2_pmsg := 'Off'; END_IF
SOP650_KM1_2_publish := _w41 OR _w42 OR _w43;

// NETWORK 22
_w44 := SOP650_KM1_2_pmsg <> SOP650_KM1_2_last_pmsg AND NOT SOP650_KM1_2_pbusy;
IF _w44 THEN SOP650_KM1_2_last_pmsg := SOP650_KM1_2_pmsg; END_IF
SOP650_KM1_2_publish := _w44;

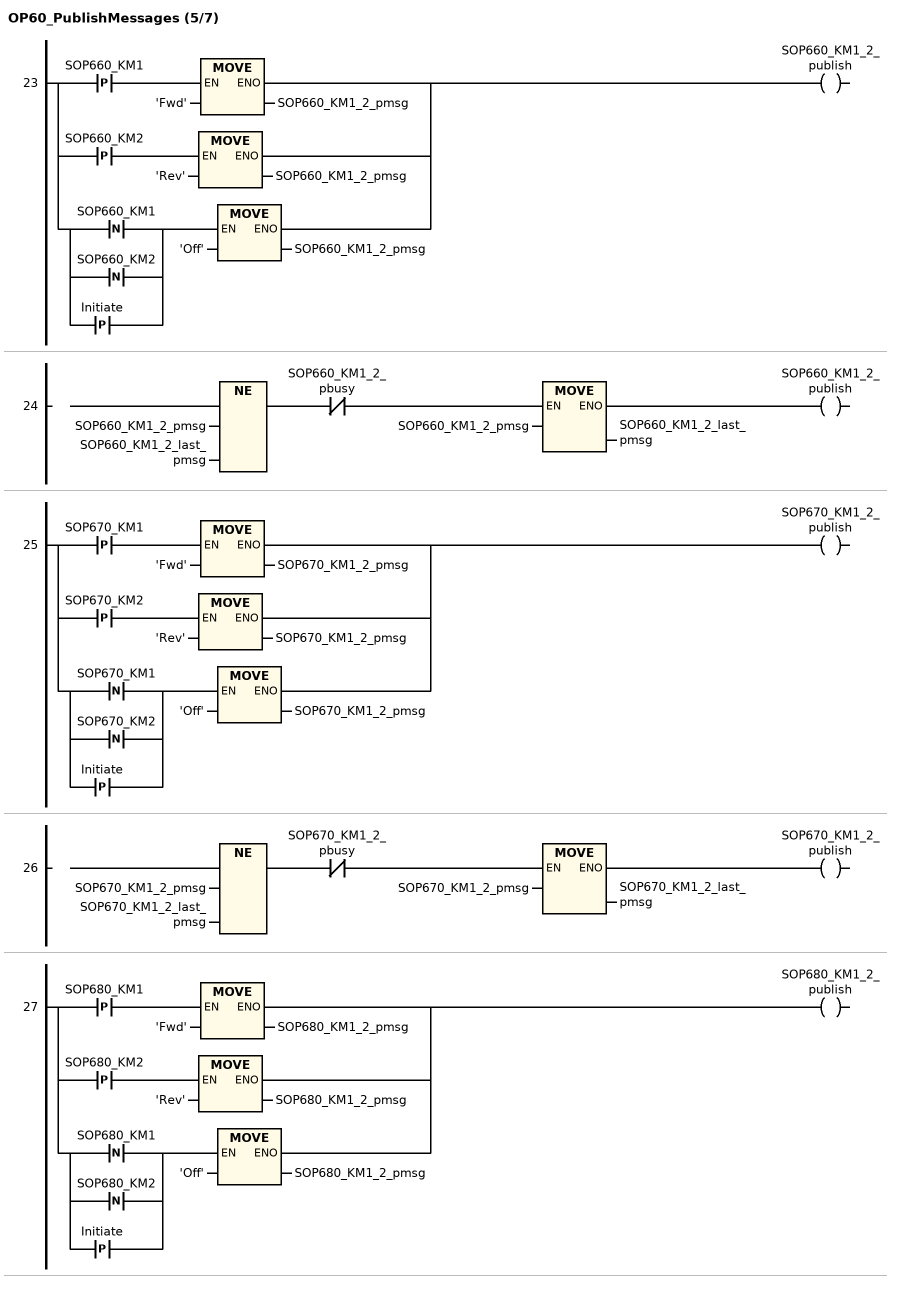
// NETWORK 23
_rt36(CLK := SOP660_KM1);
_w45 := _rt36.Q;
IF _w45 THEN SOP660_KM1_2_pmsg := 'Fwd'; END_IF
_rt37(CLK := SOP660_KM2);
_w46 := _rt37.Q;
IF _w46 THEN SOP660_KM1_2_pmsg := 'Rev'; END_IF
_ft23(CLK := SOP660_KM1);
_ft24(CLK := SOP660_KM2);
_rt38(CLK := Initiate);
_w47 := _ft23.Q OR _ft24.Q OR _rt38.Q;
IF _w47 THEN SOP660_KM1_2_pmsg := 'Off'; END_IF
SOP660_KM1_2_publish := _w45 OR _w46 OR _w47;

// NETWORK 24
_w48 := SOP660_KM1_2_pmsg <> SOP660_KM1_2_last_pmsg AND NOT SOP660_KM1_2_pbusy;
IF _w48 THEN SOP660_KM1_2_last_pmsg := SOP660_KM1_2_pmsg; END_IF
SOP660_KM1_2_publish := _w48;

// NETWORK 25
_rt39(CLK := SOP670_KM1);
_w49 := _rt39.Q;
IF _w49 THEN SOP670_KM1_2_pmsg := 'Fwd'; END_IF
_rt40(CLK := SOP670_KM2);
_w50 := _rt40.Q;
IF _w50 THEN SOP670_KM1_2_pmsg := 'Rev'; END_IF
_ft25(CLK := SOP670_KM1);
_ft26(CLK := SOP670_KM2);
_rt41(CLK := Initiate);
_w51 := _ft25.Q OR _ft26.Q OR _rt41.Q;
IF _w51 THEN SOP670_KM1_2_pmsg := 'Off'; END_IF
SOP670_KM1_2_publish := _w49 OR _w50 OR _w51;

// NETWORK 26
_w52 := SOP670_KM1_2_pmsg <> SOP670_KM1_2_last_pmsg AND NOT SOP670_KM1_2_pbusy;
IF _w52 THEN SOP670_KM1_2_last_pmsg := SOP670_KM1_2_pmsg; END_IF
SOP670_KM1_2_publish := _w52;

// NETWORK 27
_rt42(CLK := SOP680_KM1);
_w53 := _rt42.Q;
IF _w53 THEN SOP680_KM1_2_pmsg := 'Fwd'; END_IF
_rt43(CLK := SOP680_KM2);
_w54 := _rt43.Q;
IF _w54 THEN SOP680_KM1_2_pmsg := 'Rev'; END_IF
_ft27(CLK := SOP680_KM1);
_ft28(CLK := SOP680_KM2);
_rt44(CLK := Initiate);
_w55 := _ft27.Q OR _ft28.Q OR _rt44.Q;
IF _w55 THEN SOP680_KM1_2_pmsg := 'Off'; END_IF
SOP680_KM1_2_publish := _w53 OR _w54 OR _w55;

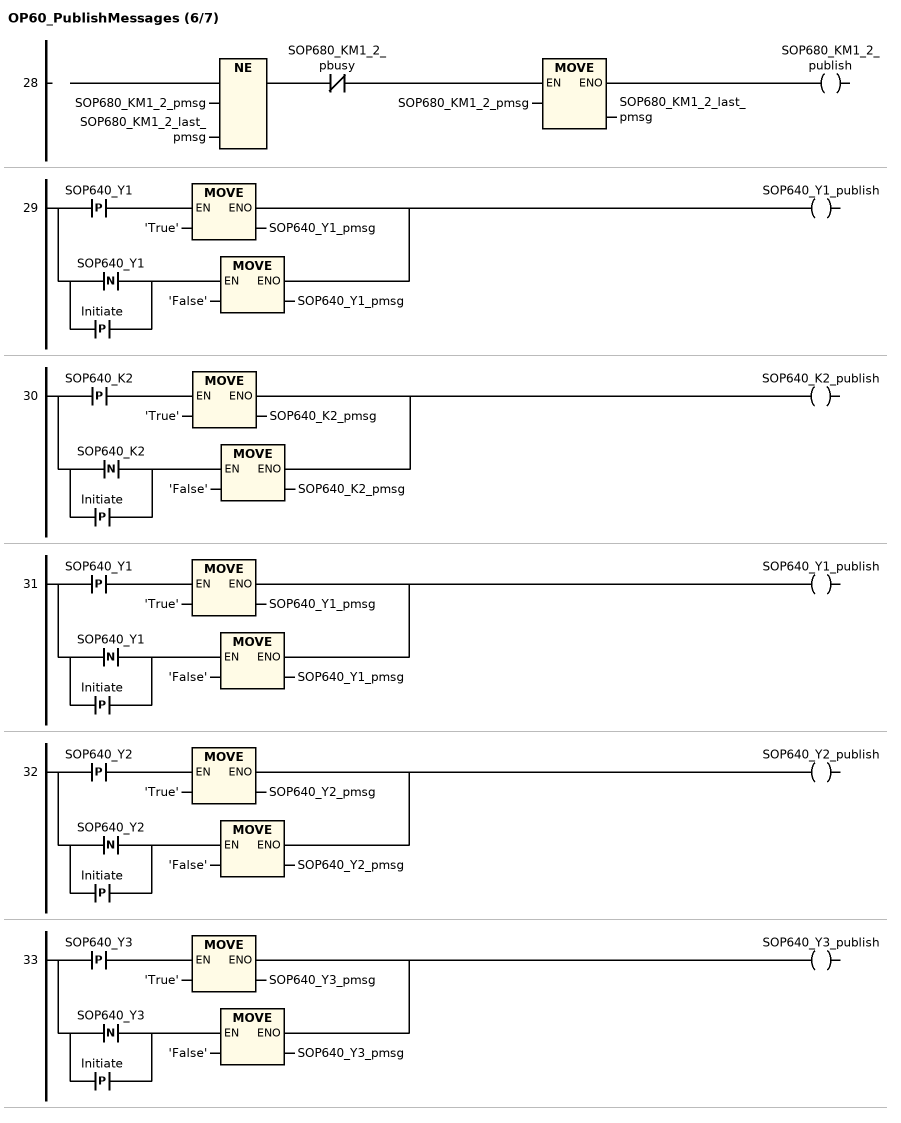
// NETWORK 28
_w56 := SOP680_KM1_2_pmsg <> SOP680_KM1_2_last_pmsg AND NOT SOP680_KM1_2_pbusy;
IF _w56 THEN SOP680_KM1_2_last_pmsg := SOP680_KM1_2_pmsg; END_IF
SOP680_KM1_2_publish := _w56;

// NETWORK 29
_rt45(CLK := SOP640_Y1);
_w57 := _rt45.Q;
IF _w57 THEN SOP640_Y1_pmsg := 'True'; END_IF
_ft29(CLK := SOP640_Y1);
_rt46(CLK := Initiate);
_w58 := _ft29.Q OR _rt46.Q;
IF _w58 THEN SOP640_Y1_pmsg := 'False'; END_IF
SOP640_Y1_publish := _w57 OR _w58;

// NETWORK 30
_rt47(CLK := SOP640_K2);
_w59 := _rt47.Q;
IF _w59 THEN SOP640_K2_pmsg := 'True'; END_IF
_ft30(CLK := SOP640_K2);
_rt48(CLK := Initiate);
_w60 := _ft30.Q OR _rt48.Q;
IF _w60 THEN SOP640_K2_pmsg := 'False'; END_IF
SOP640_K2_publish := _w59 OR _w60;

// NETWORK 31
_rt49(CLK := SOP640_Y1);
_w61 := _rt49.Q;
IF _w61 THEN SOP640_Y1_pmsg := 'True'; END_IF
_ft31(CLK := SOP640_Y1);
_rt50(CLK := Initiate);
_w62 := _ft31.Q OR _rt50.Q;
IF _w62 THEN SOP640_Y1_pmsg := 'False'; END_IF
SOP640_Y1_publish := _w61 OR _w62;

// NETWORK 32
_rt51(CLK := SOP640_Y2);
_w63 := _rt51.Q;
IF _w63 THEN SOP640_Y2_pmsg := 'True'; END_IF
_ft32(CLK := SOP640_Y2);
_rt52(CLK := Initiate);
_w64 := _ft32.Q OR _rt52.Q;
IF _w64 THEN SOP640_Y2_pmsg := 'False'; END_IF
SOP640_Y2_publish := _w63 OR _w64;

// NETWORK 33
_rt53(CLK := SOP640_Y3);
_w65 := _rt53.Q;
IF _w65 THEN SOP640_Y3_pmsg := 'True'; END_IF
_ft33(CLK := SOP640_Y3);
_rt54(CLK := Initiate);
_w66 := _ft33.Q OR _rt54.Q;
IF _w66 THEN SOP640_Y3_pmsg := 'False'; END_IF
SOP640_Y3_publish := _w65 OR _w66;

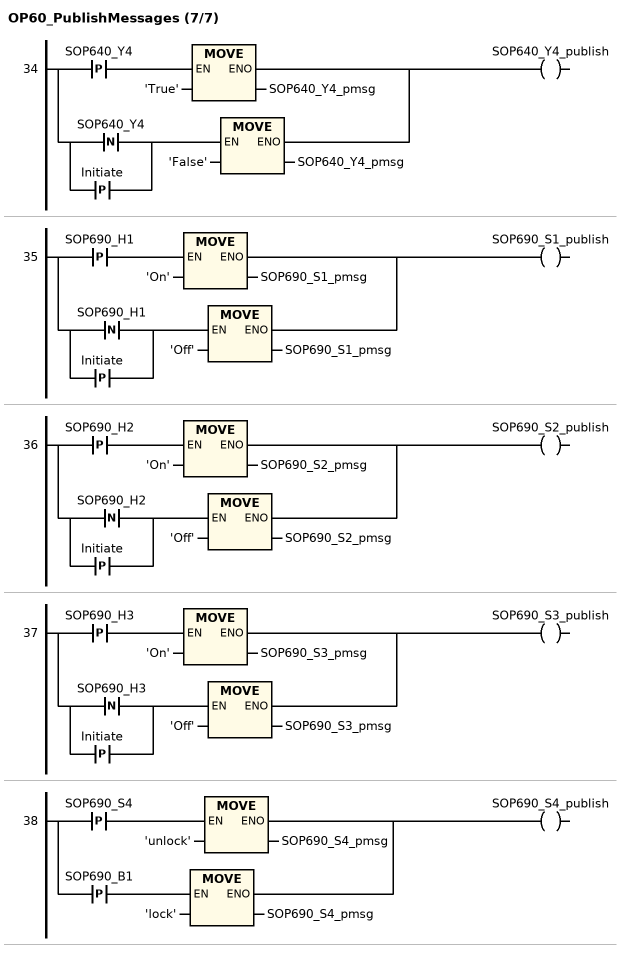
// NETWORK 34
_rt55(CLK := SOP640_Y4);
_w67 := _rt55.Q;
IF _w67 THEN SOP640_Y4_pmsg := 'True'; END_IF
_ft34(CLK := SOP640_Y4);
_rt56(CLK := Initiate);
_w68 := _ft34.Q OR _rt56.Q;
IF _w68 THEN SOP640_Y4_pmsg := 'False'; END_IF
SOP640_Y4_publish := _w67 OR _w68;

// NETWORK 35
_rt57(CLK := SOP690_H1);
_w69 := _rt57.Q;
IF _w69 THEN SOP690_S1_pmsg := 'On'; END_IF
_ft35(CLK := SOP690_H1);
_rt58(CLK := Initiate);
_w70 := _ft35.Q OR _rt58.Q;
IF _w70 THEN SOP690_S1_pmsg := 'Off'; END_IF
SOP690_S1_publish := _w69 OR _w70;

// NETWORK 36
_rt59(CLK := SOP690_H2);
_w71 := _rt59.Q;
IF _w71 THEN SOP690_S2_pmsg := 'On'; END_IF
_ft36(CLK := SOP690_H2);
_rt60(CLK := Initiate);
_w72 := _ft36.Q OR _rt60.Q;
IF _w72 THEN SOP690_S2_pmsg := 'Off'; END_IF
SOP690_S2_publish := _w71 OR _w72;

// NETWORK 37
_rt61(CLK := SOP690_H3);
_w73 := _rt61.Q;
IF _w73 THEN SOP690_S3_pmsg := 'On'; END_IF
_ft37(CLK := SOP690_H3);
_rt62(CLK := Initiate);
_w74 := _ft37.Q OR _rt62.Q;
IF _w74 THEN SOP690_S3_pmsg := 'Off'; END_IF
SOP690_S3_publish := _w73 OR _w74;

// NETWORK 38
_rt63(CLK := SOP690_S4);
_w75 := _rt63.Q;
IF _w75 THEN SOP690_S4_pmsg := 'unlock'; END_IF
_rt64(CLK := SOP690_B1);
_w76 := _rt64.Q;
IF _w76 THEN SOP690_S4_pmsg := 'lock'; END_IF
SOP690_S4_publish := _w75 OR _w76;

END_PROGRAM

// Device/Application/OP60_Illumination
PROGRAM OP60_Illumination
VAR
	enable: BOOL;
	RS_0: RS;
	Mid_signal: BOOL;
END_VAR
VAR // added by the converter: edge detectors and wires of the graphical bodies
    _w1, _w2 : BOOL;
END_VAR

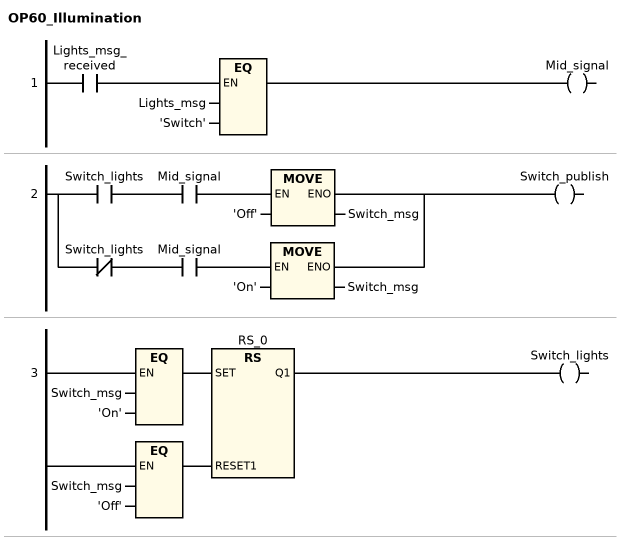
// NETWORK 1
Mid_signal := Lights_msg_received AND Lights_msg = 'Switch';

// NETWORK 2
_w1 := Switch_lights AND Mid_signal;
IF _w1 THEN Switch_msg := 'Off'; END_IF
_w2 := NOT Switch_lights AND Mid_signal;
IF _w2 THEN Switch_msg := 'On'; END_IF
Switch_publish := _w1 OR _w2;

// NETWORK 3
RS_0(SET := Switch_msg = 'On', RESET1 := Switch_msg = 'Off'); // RS
Switch_lights := RS_0.Q1;

END_PROGRAM

// Device/Application/OP60_Schedule
PROGRAM OP60_Schedule
VAR
	Change_Schedule: BOOL;
	Define_start: BOOL;
	Check_button_not_pushed: BOOL;
	Define_end: BOOL;
	SR_publish: BOOL;
	Publish_OK: BOOL;
	OP60_end: BOOL; 
	OP60_start: BOOL; 
	
	Start_time: STRING(32) := '08:00';
	End_time: STRING(32) := '20:00';
	
	RS_0: RS;
	TON_0: TON;
	TimerON_0: TIME;
	TON_1: TON;
	TimerON_1: TIME;
	TON_2: TON;
	TimerON_2: TIME;
	TON_3: TON;
	TimerON_3: TIME;
	TON_4: TON;
	TimerON_4: TIME;
	Publish_off: BOOL;
	Publish_off1: BOOL;
	Publish_off2: BOOL;
	Publish_off3: BOOL;
END_VAR
VAR // added by the converter: edge detectors and wires of the graphical bodies
    _w1 : BOOL;
END_VAR

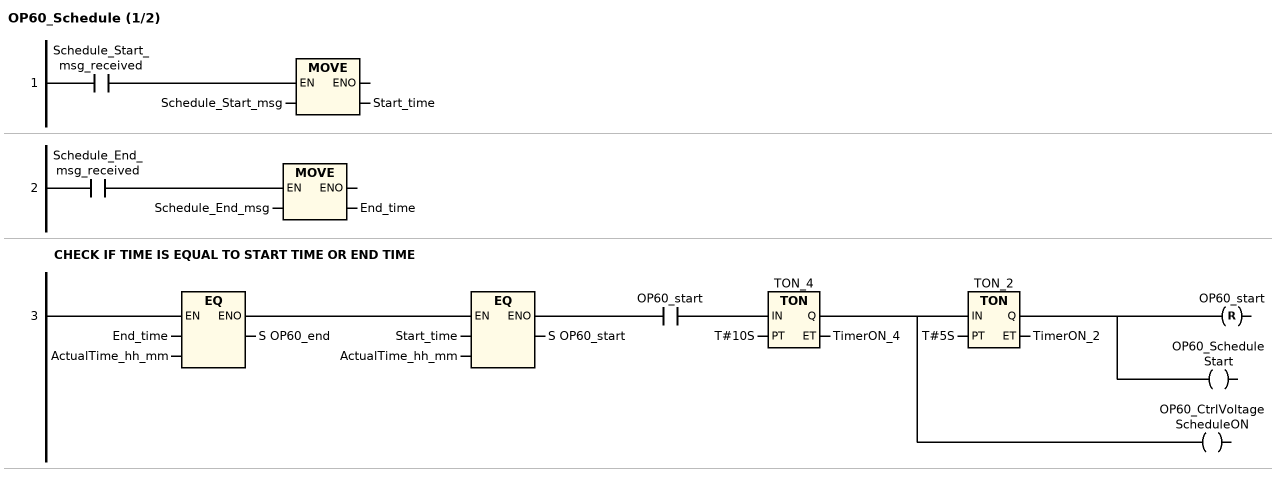
// NETWORK 1
IF Schedule_Start_msg_received THEN Start_time := Schedule_Start_msg; END_IF

// NETWORK 2
IF Schedule_End_msg_received THEN End_time := Schedule_End_msg; END_IF

// NETWORK 3: CHECK IF TIME IS EQUAL TO START TIME OR END TIME
OP60_end S= End_time = ActualTime_hh_mm;
OP60_start S= Start_time = ActualTime_hh_mm;
TON_4(IN := OP60_start, PT := T#10S, ET => TimerON_4); // TON
TON_2(IN := TON_4.Q, PT := T#5S, ET => TimerON_2); // TON
OP60_start R= TON_2.Q;
OP60_ScheduleStart := TON_2.Q;
OP60_CtrlVoltageScheduleON := TON_4.Q;

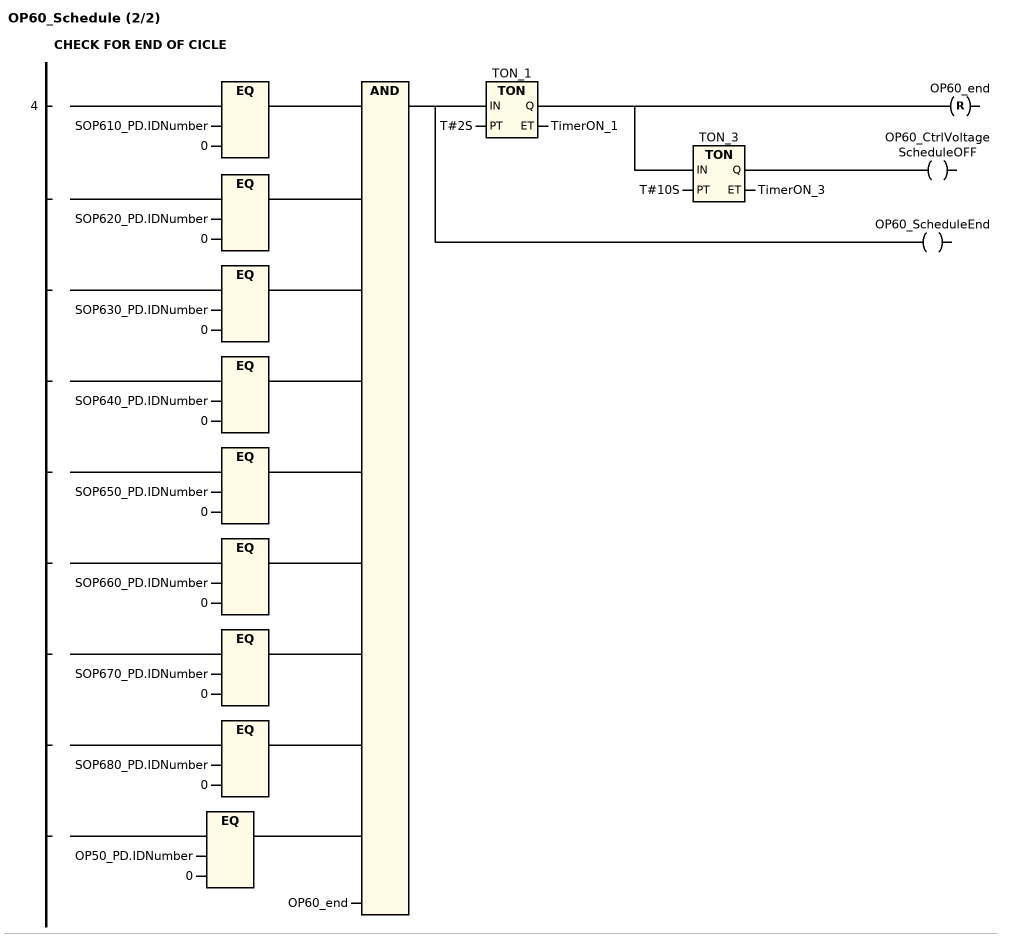
// NETWORK 4: CHECK FOR END OF CICLE
_w1 := SOP610_PD.IDNumber = 0 AND SOP620_PD.IDNumber = 0 AND SOP630_PD.IDNumber = 0 AND SOP640_PD.IDNumber = 0 AND SOP650_PD.IDNumber = 0 AND SOP660_PD.IDNumber = 0 AND SOP670_PD.IDNumber = 0 AND SOP680_PD.IDNumber = 0 AND OP50_PD.IDNumber = 0 AND OP60_end;
TON_1(IN := _w1, PT := T#2S, ET => TimerON_1); // TON
OP60_end R= TON_1.Q;
TON_3(IN := TON_1.Q, PT := T#10S, ET => TimerON_3); // TON
OP60_CtrlVoltageScheduleOFF := TON_3.Q;
OP60_ScheduleEnd := _w1;

END_PROGRAM

// Device/Application/FBs/DateAndTime
PROGRAM DateAndTime
VAR
	Date_and_time_in_seconds : UDINT;
	Local_date_time_seconds : UDINT;
	Date_and_Time_result : UDINT;
	Local_date_time_from_secs : SYSTIMEDATE;
	Date_and_time_format : DATE_AND_TIME;
	Date_and_time_string : STRING;
END_VAR

// Get TIME in seconds since 1970 :
Date_and_time_in_seconds := SysTimeRtcGet(Date_and_Time_result);
IF Date_and_Time_result <> 0 THEN
RETURN;
END_IF

// Convert UTC seconds to local time seconds, regarding Timezone and Summer time :
Date_and_Time_result := SysTimeRtcConvertUtcToLocal(Date_and_time_in_seconds, Local_date_time_seconds);
IF Date_and_Time_result <> 0 THEN
RETURN;
END_IF

// Convert the UTC seconds to a DATE_AND_TIME variable dt#yyyy-mm-dd-hh:mm:ss :
Date_and_time_format := UDINT_TO_DT(Local_date_time_seconds);

// Convert DATE_AND_TIME to a String :
Date_and_time_string := DT_TO_STRING(Date_and_time_format);
ActualTime_hh_mm_ss := RIGHT(Date_and_time_string, 8);
ActualTime_hh_mm := LEFT(ActualTime_hh_mm_ss,5);

END_PROGRAM

// Device/Application/SOP680
PROGRAM SOP680
VAR
END_VAR
VAR // added by the converter: edge detectors and wires of the graphical bodies
    _rt1 : R_TRIG;
END_VAR

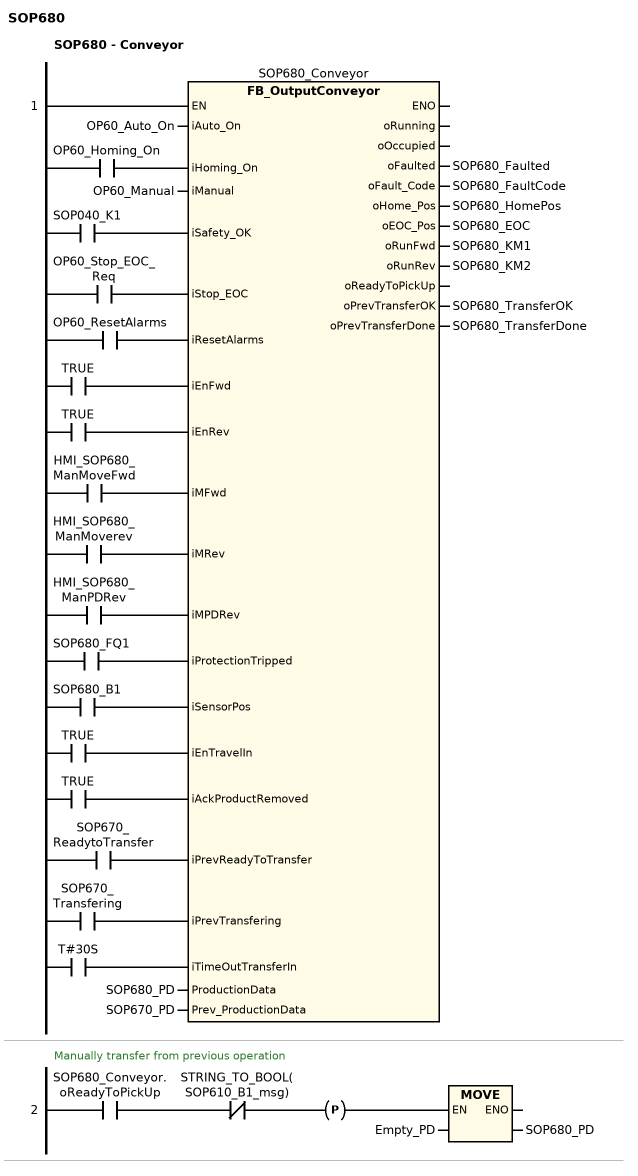
// NETWORK 1: SOP680 - Conveyor
SOP680_Conveyor(
    iAuto_On := OP60_Auto_On,
    iHoming_On := OP60_Homing_On,
    iManual := OP60_Manual,
    iSafety_OK := SOP040_K1,
    iStop_EOC := OP60_Stop_EOC_Req,
    iResetAlarms := OP60_ResetAlarms,
    iEnFwd := TRUE,
    iEnRev := TRUE,
    iMFwd := HMI_SOP680_ManMoveFwd,
    iMRev := HMI_SOP680_ManMoverev,
    iMPDRev := HMI_SOP680_ManPDRev,
    iProtectionTripped := SOP680_FQ1,
    iSensorPos := SOP680_B1,
    iEnTravelIn := TRUE,
    iAckProductRemoved := TRUE,
    iPrevReadyToTransfer := SOP670_ReadytoTransfer,
    iPrevTransfering := SOP670_Transfering,
    iTimeOutTransferIn := T#30S,
    ProductionData := SOP680_PD,
    Prev_ProductionData := SOP670_PD,
    oFaulted => SOP680_Faulted,
    oFault_Code => SOP680_FaultCode,
    oHome_Pos => SOP680_HomePos,
    oEOC_Pos => SOP680_EOC,
    oRunFwd => SOP680_KM1,
    oRunRev => SOP680_KM2,
    oPrevTransferOK => SOP680_TransferOK,
    oPrevTransferDone => SOP680_TransferDone); // FB_OutputConveyor

// NETWORK 2
// Manually transfer from previous operation
_rt1(CLK := SOP680_Conveyor.oReadyToPickUp AND NOT (STRING_TO_BOOL(SOP610_B1_msg)));
IF _rt1.Q THEN SOP680_PD := Empty_PD; END_IF

END_PROGRAM

// Device/Application/FBs/FB_OutputConveyor
FUNCTION_BLOCK FB_OutputConveyor
VAR_INPUT
	iAuto_On: BOOL; // Auto-On cycle active
	iHoming_On: BOOL; // Homing-On cycle active
	iManual: BOOL; // Manual mode active
	iSafety_OK: BOOL; // Safety circuit OK
	iStop_EOC: BOOL; // Stop EOC selected
	iResetAlarms: BOOL; // Reset Alarms
	
	iEnFwd: BOOL := TRUE; // Interlock signal movement forward
	iEnRev: BOOL := TRUE; // Interlock signal movement reverse
	
	iMFwd: BOOL; 	// Manual Fwd request
	iMRev: BOOL; 	// Manual Rev request
	iMPDRev: BOOL; 	// Manual Move PD reverse
	
	iProtectionTripped: BOOL := FALSE; // Motor Protection Tripped
	
	iSensorPos: BOOL; // Product in position
	
	iEnTravelIn: BOOL := TRUE; // Enable product transfer from previous conveyor.
	iAckProductRemoved: BOOL := FALSE; // ACknowledge product has been removed from the conveyor.
	
	iPrevReadyToTransfer: BOOL; // Previous conveyor ready to transfer
	iPrevTransfering: BOOL; // Previous conveyor transfering
	
	iTimeOutTransferIn: TIME := T#10S; // Time out time for transfer in
END_VAR
VAR_IN_OUT
	ProductionData: ProductionData; 		// Production Data
	Prev_ProductionData: ProductionData;	// Previous Production Data
END_VAR
VAR_OUTPUT
	oRunning: BOOL; // Conveyor Running
	oOccupied: BOOL; // Conveyor Occupied
	oFaulted : BOOL; // Conveyor faulted
	oFault_Code: INT; // Conveyor fault code
	oHome_Pos: BOOL; // Conveyor Home Position reached
	oEOC_Pos: BOOL; // Conveyor Stop EOC reached

	oRunFwd: BOOL; // Conveyor running forward
	oRunRev: BOOL; // Conveyor running reverse	

	oReadyToPickUp: BOOL; // Conveyor ready to pick up
	oPrevTransferOK: BOOL; // Conveyor ready to load
	oPrevTransferDone: BOOL; // Conveyor load completed
END_VAR
VAR
	AutoSteps: WORD;
	HomeSteps: WORD;
	
	Timeout_Fault1: TON;
	
	EmptyPD: ProductionData;
	PDValid: BOOL;		// PD is Valid
	PDEmpty: BOOL;		// PD is Empty
	PrevPDValid: BOOL;	// Previous PD is Valid
	PrevPDEmpty: BOOL;	// Previous PD is Empty
	R_TRIG_TransferPDRev: R_TRIG;
	R_TRIG_Fault_11: R_TRIG;
	R_TRIG_Fault_12: R_TRIG;
END_VAR
VAR // added by the converter: edge detectors and wires of the graphical bodies
    _w1, _w2, _w3, _w4, _w5, _w6, _w7, _w8, _w9, _w10, _w11, _w12, _w13 : BOOL;
END_VAR

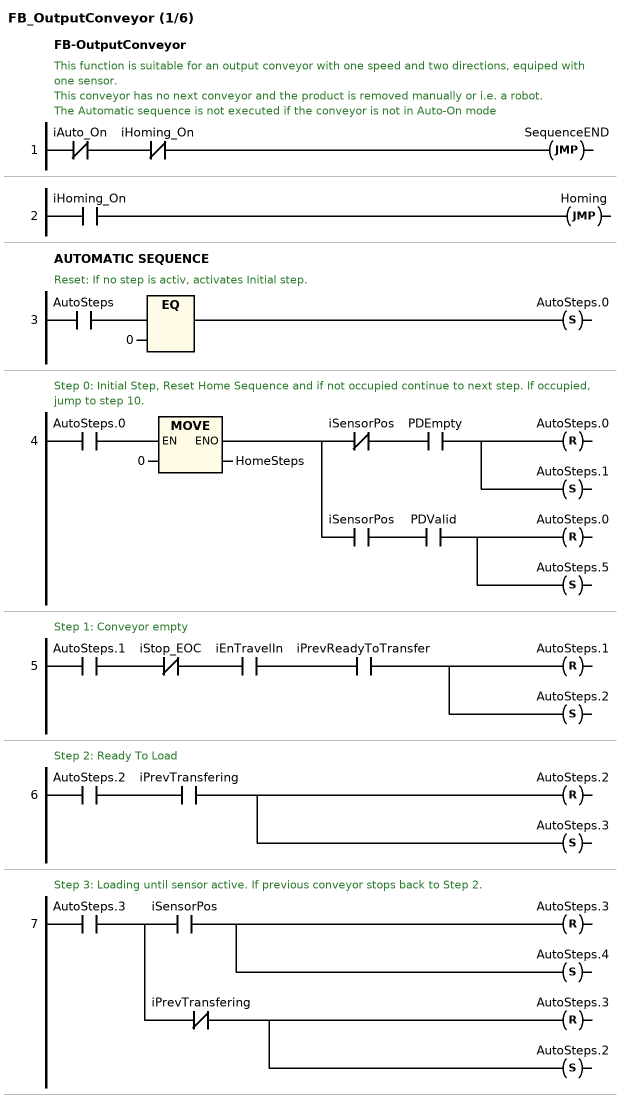
// NETWORK 1: FB-OutputConveyor
// This function is suitable for an output conveyor with one speed and two directions, equiped with one sensor.
// This conveyor has no next conveyor and the product is removed manually or i.e. a robot.
// The Automatic sequence is not executed if the conveyor is not in Auto-On mode
IF NOT iAuto_On AND NOT iHoming_On THEN JMP SequenceEND; END_IF

// NETWORK 2
IF iHoming_On THEN JMP Homing; END_IF

// NETWORK 3: AUTOMATIC SEQUENCE
// Reset: If no step is activ, activates Initial step.
AutoSteps.0 S= AutoSteps = 0;

// NETWORK 4
// Step 0: Initial Step, Reset Home Sequence and if not occupied continue to next step. If occupied, jump to step 10.
_w1 := AutoSteps.0;
IF _w1 THEN HomeSteps := 0; END_IF
_w2 := _w1 AND NOT iSensorPos AND PDEmpty;
AutoSteps.0 R= _w2;
AutoSteps.1 S= _w2;
_w3 := _w1 AND iSensorPos AND PDValid;
AutoSteps.0 R= _w3;
AutoSteps.5 S= _w3;

// NETWORK 5
// Step 1: Conveyor empty
_w4 := AutoSteps.1 AND NOT iStop_EOC AND iEnTravelIn AND iPrevReadyToTransfer;
AutoSteps.1 R= _w4;
AutoSteps.2 S= _w4;

// NETWORK 6
// Step 2: Ready To Load
_w5 := AutoSteps.2 AND iPrevTransfering;
AutoSteps.2 R= _w5;
AutoSteps.3 S= _w5;

// NETWORK 7
// Step 3: Loading until sensor active. If previous conveyor stops back to Step 2.
_w6 := AutoSteps.3;
_w7 := _w6 AND iSensorPos;
AutoSteps.3 R= _w7;
AutoSteps.4 S= _w7;
_w8 := _w6 AND NOT iPrevTransfering;
AutoSteps.3 R= _w8;
AutoSteps.2 S= _w8;

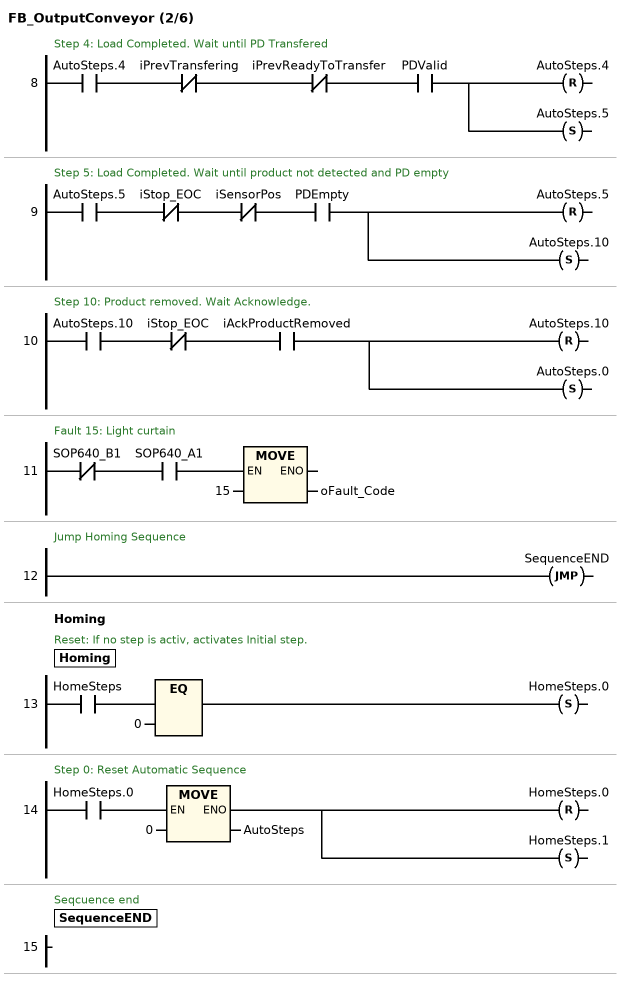
// NETWORK 8
// Step 4: Load Completed. Wait until PD Transfered
_w9 := AutoSteps.4 AND NOT iPrevTransfering AND NOT iPrevReadyToTransfer AND PDValid;
AutoSteps.4 R= _w9;
AutoSteps.5 S= _w9;

// NETWORK 9
// Step 5: Load Completed. Wait until product not detected and PD empty
_w10 := AutoSteps.5 AND NOT iStop_EOC AND NOT iSensorPos AND PDEmpty;
AutoSteps.5 R= _w10;
AutoSteps.10 S= _w10;

// NETWORK 10
// Step 10: Product removed. Wait Acknowledge.
_w11 := AutoSteps.10 AND NOT iStop_EOC AND iAckProductRemoved;
AutoSteps.10 R= _w11;
AutoSteps.0 S= _w11;

// NETWORK 11
// Fault 15: Light curtain
IF NOT SOP640_B1 AND SOP640_A1 THEN oFault_Code := 15; END_IF

// NETWORK 12
// Jump Homing Sequence
JMP SequenceEND;

// NETWORK 13: Homing
// Reset: If no step is activ, activates Initial step.
Homing:
HomeSteps.0 S= HomeSteps = 0;

// NETWORK 14
// Step 0: Reset Automatic Sequence
_w12 := HomeSteps.0;
IF _w12 THEN AutoSteps := 0; END_IF
HomeSteps.0 R= _w12;
HomeSteps.1 S= _w12;

// NETWORK 15
// Seqcuence end
SequenceEND: ;

